REGION Network 21: bit gotowości wspólny Z9
   // AUMA
   // MODACT MOK250
   RUNG wire#powerrail
      Contact( "AlwaysTRUE" )
      Contact( "isPowerOK" )
      wire#w1
      Contact( "isAUMA_Z_9" )
      I_Contact( "inputAumagotowośćZ_9" )
      wire#w2
      R_Coil( "isGotowość_Z_9" )
   END_RUNG
   RUNG wire#w1
      Contact( "Hbit_Alarm_Z9" )
   END_RUNG wire#w2
   RUNG wire#w1
      I_Contact( "isAUMA_Z_9" )
      Contact( "setAlarm_Moment_Z_9" )
   END_RUNG wire#w2
   RUNG wire#w1
      Contact( "Hbit_Alarm_Z9" )
      Coil( "CMD_Awaria_Z_9" )
   END_RUNG
   // the same network as SCL:
   #_w1 := "AlwaysTRUE" AND "isPowerOK";
   IF #_w1 AND (("isAUMA_Z_9" AND NOT "inputAumagotowośćZ_9") OR "Hbit_Alarm_Z9" OR (NOT "isAUMA_Z_9" AND "setAlarm_Moment_Z_9")) THEN
       "isGotowość_Z_9" := FALSE;
   END_IF;
   "CMD_Awaria_Z_9" := #_w1 AND "Hbit_Alarm_Z9";
END_REGION
END_FUNCTION

FUNCTION "Wybór_aktywnego_zbiornika" : Void   // FC20, LAD
TITLE = Compressor selection from hours
{ S7_Optimized_Access := 'TRUE' }
AUTHOR : rtecmer
VERSION : 0.1
// Ustawienie kolejności wyboru zbiornika z wyrównaniem czasu pracy. Podstawa najmniejsza ilość godzin pracy
// stored: AutoNumber true, IsIECCheckEnabled false, SetENOAutomatically false, UDAEnableTagReadback false
   VAR_INPUT
      aktywny_Zbiornik_1 : Bool;   // zbiornik aktywny zasuwy na pozycji atomat
      aktywny_Zbiornik_2 : Bool;
      aktywny_Zbiornik_3 : Bool;
      aktywny_Zbiornik_4 : Bool;
      ready_Z1 : Bool;   // gotowość
      ready_Z2 : Bool;   // gotowość
      ready_Z3 : Bool;   // gotowość
      ready_Z4 : Bool;   // gotowość
      ready_Z5 : Bool;   // gotowość
      ready_Z6 : Bool;   // gotowość
      ready_Z7 : Bool;   // gotowość
      ready_Z8 : Bool;   // gotowość
      Is_Eptying : Bool;   // aktwny cykl napełniania
      Is_Filling : Bool;   // aktywny cykl pompownia
   END_VAR
   VAR_IN_OUT
      Reset : Bool;   // Reset po błędzie
      set_HWork_Tank_1 : Bool;   // ustawiony aktywny
      set_HWork_Tank_2 : Bool;   // ustawiony aktywny
      set_HWork_Tank_3 : Bool;   // ustawiony aktywny
      set_HWork_Tank_4 : Bool;   // ustawiony aktywny
      blok_tank_1 : Bool;   // blokowanie zbirnika w sekwencji
      blok_tank_2 : Bool;   // blokowanie zbirnika w sekwencji
      blok_tank_3 : Bool;   // blokowanie zbirnika w sekwencji
      blok_tank_4 : Bool;   // blokowanie zbirnika w sekwencji
   END_VAR
   VAR_TEMP
      tmp_Sum_sek_P1 : Real;
      tmp_Sum_sek_P2 : Real;
      tmp_Sum_sek_P3 : Real;
      tmp_Sum_sek_P4 : Real;
   END_VAR
BEGIN

REGION Network 1: Reakcja na równe liczniki
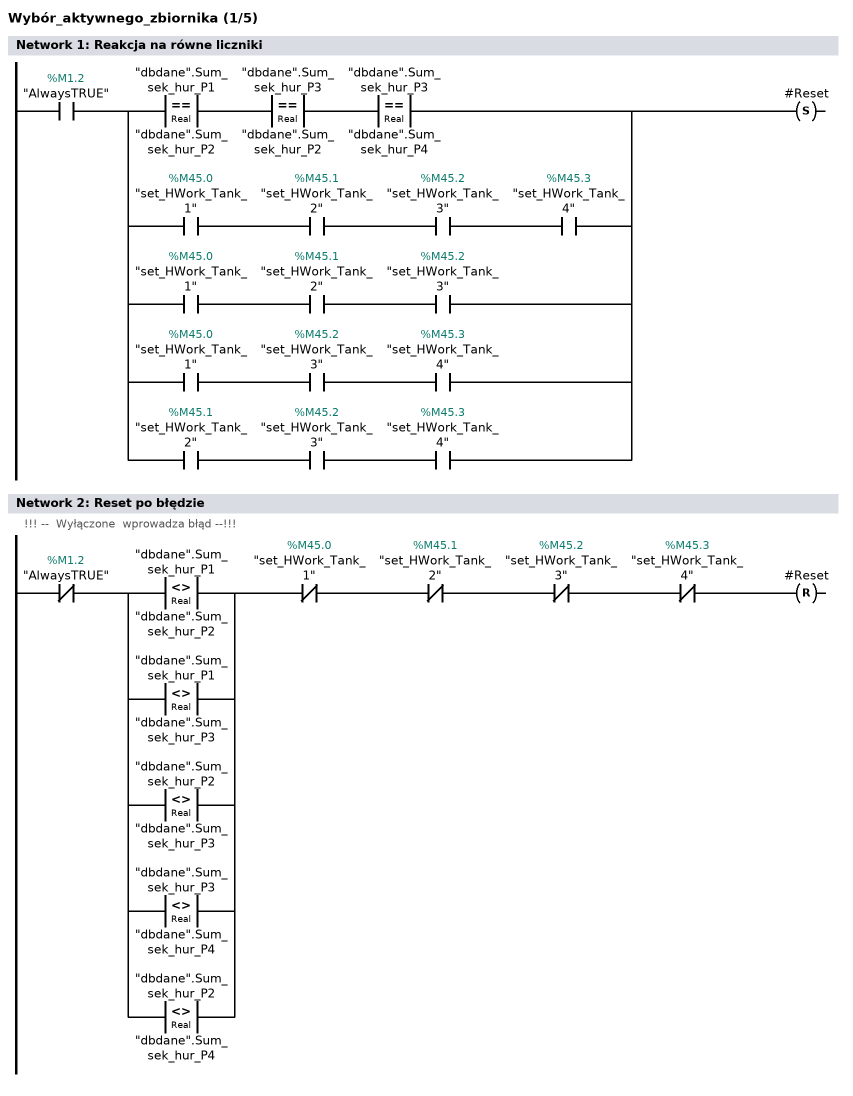
   RUNG wire#powerrail
      Contact( "AlwaysTRUE" )
      wire#w1
      { S7_Templates := "SrcType := Real" } EQ_Contact(in1 := "dbdane".Sum_sek_hur_P1, in2 := "dbdane".Sum_sek_hur_P2)
      { S7_Templates := "SrcType := Real" } EQ_Contact(in1 := "dbdane".Sum_sek_hur_P3, in2 := "dbdane".Sum_sek_hur_P2)
      { S7_Templates := "SrcType := Real" } EQ_Contact(in1 := "dbdane".Sum_sek_hur_P3, in2 := "dbdane".Sum_sek_hur_P4)
      wire#w2
      S_Coil( #Reset )
   END_RUNG
   RUNG wire#w1
      Contact( "set_HWork_Tank_1" )
      Contact( "set_HWork_Tank_2" )
      Contact( "set_HWork_Tank_3" )
      Contact( "set_HWork_Tank_4" )
   END_RUNG wire#w2
   RUNG wire#w1
      Contact( "set_HWork_Tank_1" )
      Contact( "set_HWork_Tank_2" )
      Contact( "set_HWork_Tank_3" )
   END_RUNG wire#w2
   RUNG wire#w1
      Contact( "set_HWork_Tank_1" )
      Contact( "set_HWork_Tank_3" )
      Contact( "set_HWork_Tank_4" )
   END_RUNG wire#w2
   RUNG wire#w1
      Contact( "set_HWork_Tank_2" )
      Contact( "set_HWork_Tank_3" )
      Contact( "set_HWork_Tank_4" )
   END_RUNG wire#w2
   // the same network as SCL:
   IF "AlwaysTRUE" AND ((("dbdane".Sum_sek_hur_P1 = "dbdane".Sum_sek_hur_P2) AND ("dbdane".Sum_sek_hur_P3 = "dbdane".Sum_sek_hur_P2) AND ("dbdane".Sum_sek_hur_P3 = "dbdane".Sum_sek_hur_P4)) OR ("set_HWork_Tank_1" AND "set_HWork_Tank_2" AND "set_HWork_Tank_3" AND "set_HWork_Tank_4") OR ("set_HWork_Tank_1" AND "set_HWork_Tank_2" AND "set_HWork_Tank_3") OR ("set_HWork_Tank_1" AND "set_HWork_Tank_3" AND "set_HWork_Tank_4") OR ("set_HWork_Tank_2" AND "set_HWork_Tank_3" AND "set_HWork_Tank_4")) THEN
       #Reset := TRUE;
   END_IF;
END_REGION

REGION Network 2: Reset po błędzie
   // !!! --  Wyłączone  wprowadza błąd --!!!
   RUNG wire#powerrail
      I_Contact( "AlwaysTRUE" )
      wire#w1
      { S7_Templates := "SrcType := Real" } NE_Contact(in1 := "dbdane".Sum_sek_hur_P1, in2 := "dbdane".Sum_sek_hur_P2)
      wire#w2
      I_Contact( "set_HWork_Tank_1" )
      I_Contact( "set_HWork_Tank_2" )
      I_Contact( "set_HWork_Tank_3" )
      I_Contact( "set_HWork_Tank_4" )
      R_Coil( #Reset )
   END_RUNG
   RUNG wire#w1
      { S7_Templates := "SrcType := Real" } NE_Contact(in1 := "dbdane".Sum_sek_hur_P1, in2 := "dbdane".Sum_sek_hur_P3)
   END_RUNG wire#w2
   RUNG wire#w1
      { S7_Templates := "SrcType := Real" } NE_Contact(in1 := "dbdane".Sum_sek_hur_P2, in2 := "dbdane".Sum_sek_hur_P3)
   END_RUNG wire#w2
   RUNG wire#w1
      { S7_Templates := "SrcType := Real" } NE_Contact(in1 := "dbdane".Sum_sek_hur_P3, in2 := "dbdane".Sum_sek_hur_P4)
   END_RUNG wire#w2
   RUNG wire#w1
      { S7_Templates := "SrcType := Real" } NE_Contact(in1 := "dbdane".Sum_sek_hur_P2, in2 := "dbdane".Sum_sek_hur_P4)
   END_RUNG wire#w2
   // the same network as SCL:
   IF NOT "AlwaysTRUE" AND (("dbdane".Sum_sek_hur_P1 <> "dbdane".Sum_sek_hur_P2) OR ("dbdane".Sum_sek_hur_P1 <> "dbdane".Sum_sek_hur_P3) OR ("dbdane".Sum_sek_hur_P2 <> "dbdane".Sum_sek_hur_P3) OR ("dbdane".Sum_sek_hur_P3 <> "dbdane".Sum_sek_hur_P4) OR ("dbdane".Sum_sek_hur_P2 <> "dbdane".Sum_sek_hur_P4)) AND NOT "set_HWork_Tank_1" AND NOT "set_HWork_Tank_2" AND NOT "set_HWork_Tank_3" AND NOT "set_HWork_Tank_4" THEN
       #Reset := FALSE;
   END_IF;
END_REGION

REGION Network 3: Wyłączenie napedów od równych liczników
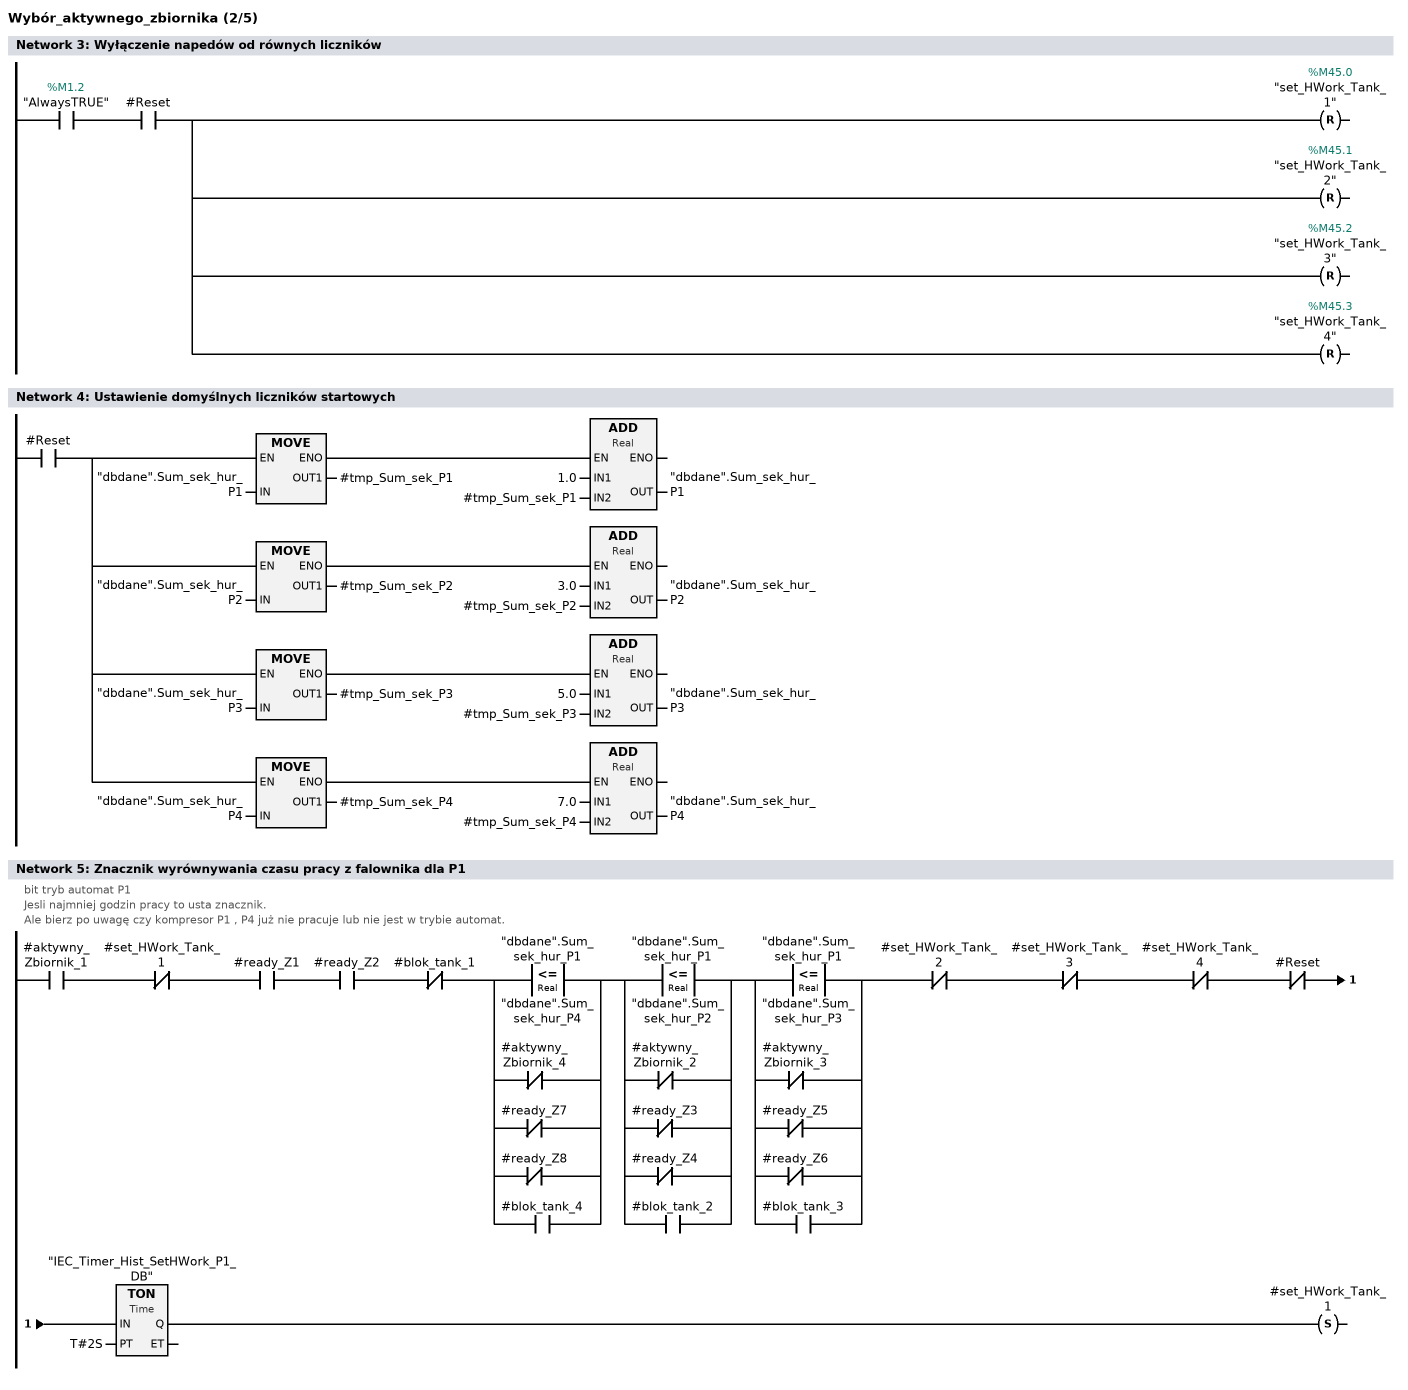
   RUNG wire#powerrail
      Contact( "AlwaysTRUE" )
      Contact( #Reset )
      wire#w1
      R_Coil( "set_HWork_Tank_1" )
   END_RUNG
   RUNG wire#w1
      R_Coil( "set_HWork_Tank_2" )
   END_RUNG
   RUNG wire#w1
      R_Coil( "set_HWork_Tank_3" )
   END_RUNG
   RUNG wire#w1
      R_Coil( "set_HWork_Tank_4" )
   END_RUNG
   // the same network as SCL:
   IF "AlwaysTRUE" AND #Reset THEN
       "set_HWork_Tank_1" := FALSE;
       "set_HWork_Tank_2" := FALSE;
       "set_HWork_Tank_3" := FALSE;
       "set_HWork_Tank_4" := FALSE;
   END_IF;
END_REGION

REGION Network 4: Ustawienie domyślnych liczników startowych
   RUNG wire#powerrail
      Contact( #Reset )
      wire#w1
      Move(in := "dbdane".Sum_sek_hur_P1, out1 => #tmp_Sum_sek_P1)
      { S7_Templates := "SrcType := Real" } Add(in1 := 1.0, in2 := #tmp_Sum_sek_P1, out => "dbdane".Sum_sek_hur_P1)
   END_RUNG
   RUNG wire#w1
      Move(in := "dbdane".Sum_sek_hur_P2, out1 => #tmp_Sum_sek_P2)
      { S7_Templates := "SrcType := Real" } Add(in1 := 3.0, in2 := #tmp_Sum_sek_P2, out => "dbdane".Sum_sek_hur_P2)
   END_RUNG
   RUNG wire#w1
      Move(in := "dbdane".Sum_sek_hur_P3, out1 => #tmp_Sum_sek_P3)
      { S7_Templates := "SrcType := Real" } Add(in1 := 5.0, in2 := #tmp_Sum_sek_P3, out => "dbdane".Sum_sek_hur_P3)
   END_RUNG
   RUNG wire#w1
      Move(in := "dbdane".Sum_sek_hur_P4, out1 => #tmp_Sum_sek_P4)
      { S7_Templates := "SrcType := Real" } Add(in1 := 7.0, in2 := #tmp_Sum_sek_P4, out => "dbdane".Sum_sek_hur_P4)
   END_RUNG
   // the same network as SCL:
   IF #Reset THEN
       #tmp_Sum_sek_P1 := "dbdane".Sum_sek_hur_P1;
       "dbdane".Sum_sek_hur_P1 := 1.0 + #tmp_Sum_sek_P1;
       #tmp_Sum_sek_P2 := "dbdane".Sum_sek_hur_P2;
       "dbdane".Sum_sek_hur_P2 := 3.0 + #tmp_Sum_sek_P2;
       #tmp_Sum_sek_P3 := "dbdane".Sum_sek_hur_P3;
       "dbdane".Sum_sek_hur_P3 := 5.0 + #tmp_Sum_sek_P3;
       #tmp_Sum_sek_P4 := "dbdane".Sum_sek_hur_P4;
       "dbdane".Sum_sek_hur_P4 := 7.0 + #tmp_Sum_sek_P4;
   END_IF;
END_REGION

REGION Network 5: Znacznik wyrównywania czasu pracy z falownika dla P1
   // bit tryb automat P1
   // Jesli najmniej godzin pracy to usta znacznik.
   // Ale bierz po uwagę czy kompresor P1 , P4 już nie pracuje lub nie jest w trybie automat.
   RUNG wire#powerrail
      Contact( #aktywny_Zbiornik_1 )
      I_Contact( #set_HWork_Tank_1 )
      Contact( #ready_Z1 )
      Contact( #ready_Z2 )
      I_Contact( #blok_tank_1 )
      wire#w1
      { S7_Templates := "SrcType := Real" } LE_Contact(in1 := "dbdane".Sum_sek_hur_P1, in2 := "dbdane".Sum_sek_hur_P4)
      wire#w2
      { S7_Templates := "SrcType := Real" } LE_Contact(in1 := "dbdane".Sum_sek_hur_P1, in2 := "dbdane".Sum_sek_hur_P2)
      wire#w3
      { S7_Templates := "SrcType := Real" } LE_Contact(in1 := "dbdane".Sum_sek_hur_P1, in2 := "dbdane".Sum_sek_hur_P3)
      wire#w4
      I_Contact( #set_HWork_Tank_2 )
      I_Contact( #set_HWork_Tank_3 )
      I_Contact( #set_HWork_Tank_4 )
      I_Contact( #Reset )
      { S7_Templates := "time_type := Time" } "IEC_Timer_Hist_SetHWork_P1_DB".TON(pt := T#2S, et =>)
      S_Coil( #set_HWork_Tank_1 )
   END_RUNG
   RUNG wire#w1
      I_Contact( #aktywny_Zbiornik_4 )
   END_RUNG wire#w2
   RUNG wire#w1
      I_Contact( #ready_Z7 )
   END_RUNG wire#w2
   RUNG wire#w1
      I_Contact( #ready_Z8 )
   END_RUNG wire#w2
   RUNG wire#w1
      Contact( #blok_tank_4 )
   END_RUNG wire#w2
   RUNG wire#w2
      I_Contact( #aktywny_Zbiornik_2 )
   END_RUNG wire#w3
   RUNG wire#w2
      I_Contact( #ready_Z3 )
   END_RUNG wire#w3
   RUNG wire#w2
      I_Contact( #ready_Z4 )
   END_RUNG wire#w3
   RUNG wire#w2
      Contact( #blok_tank_2 )
   END_RUNG wire#w3
   RUNG wire#w3
      I_Contact( #aktywny_Zbiornik_3 )
   END_RUNG wire#w4
   RUNG wire#w3
      I_Contact( #ready_Z5 )
   END_RUNG wire#w4
   RUNG wire#w3
      I_Contact( #ready_Z6 )
   END_RUNG wire#w4
   RUNG wire#w3
      Contact( #blok_tank_3 )
   END_RUNG wire#w4
   // the same network as SCL:
   "IEC_Timer_Hist_SetHWork_P1_DB".TON(IN := #aktywny_Zbiornik_1 AND NOT #set_HWork_Tank_1 AND #ready_Z1 AND #ready_Z2 AND NOT #blok_tank_1 AND (("dbdane".Sum_sek_hur_P1 <= "dbdane".Sum_sek_hur_P4) OR NOT #aktywny_Zbiornik_4 OR NOT #ready_Z7 OR NOT #ready_Z8 OR #blok_tank_4) AND (("dbdane".Sum_sek_hur_P1 <= "dbdane".Sum_sek_hur_P2) OR NOT #aktywny_Zbiornik_2 OR NOT #ready_Z3 OR NOT #ready_Z4 OR #blok_tank_2) AND (("dbdane".Sum_sek_hur_P1 <= "dbdane".Sum_sek_hur_P3) OR NOT #aktywny_Zbiornik_3 OR NOT #ready_Z5 OR NOT #ready_Z6 OR #blok_tank_3) AND NOT #set_HWork_Tank_2 AND NOT #set_HWork_Tank_3 AND NOT #set_HWork_Tank_4 AND NOT #Reset,
                           PT := T#2S);
   IF "IEC_Timer_Hist_SetHWork_P1_DB".Q THEN #set_HWork_Tank_1 := TRUE; END_IF;
END_REGION

REGION Network 6 (SCL): Sprawdzanie czy aktywna w trybie AUT
   IF "set_HWork_Tank_1" = TRUE AND #aktywny_Zbiornik_1 = FALSE THEN
     // Statement section IF
     "set_HWork_Tank_1" := FALSE;
     ;
   END_IF;
END_REGION

REGION Network 7: Znacznik ustawienia pracy od licznika pracy P1
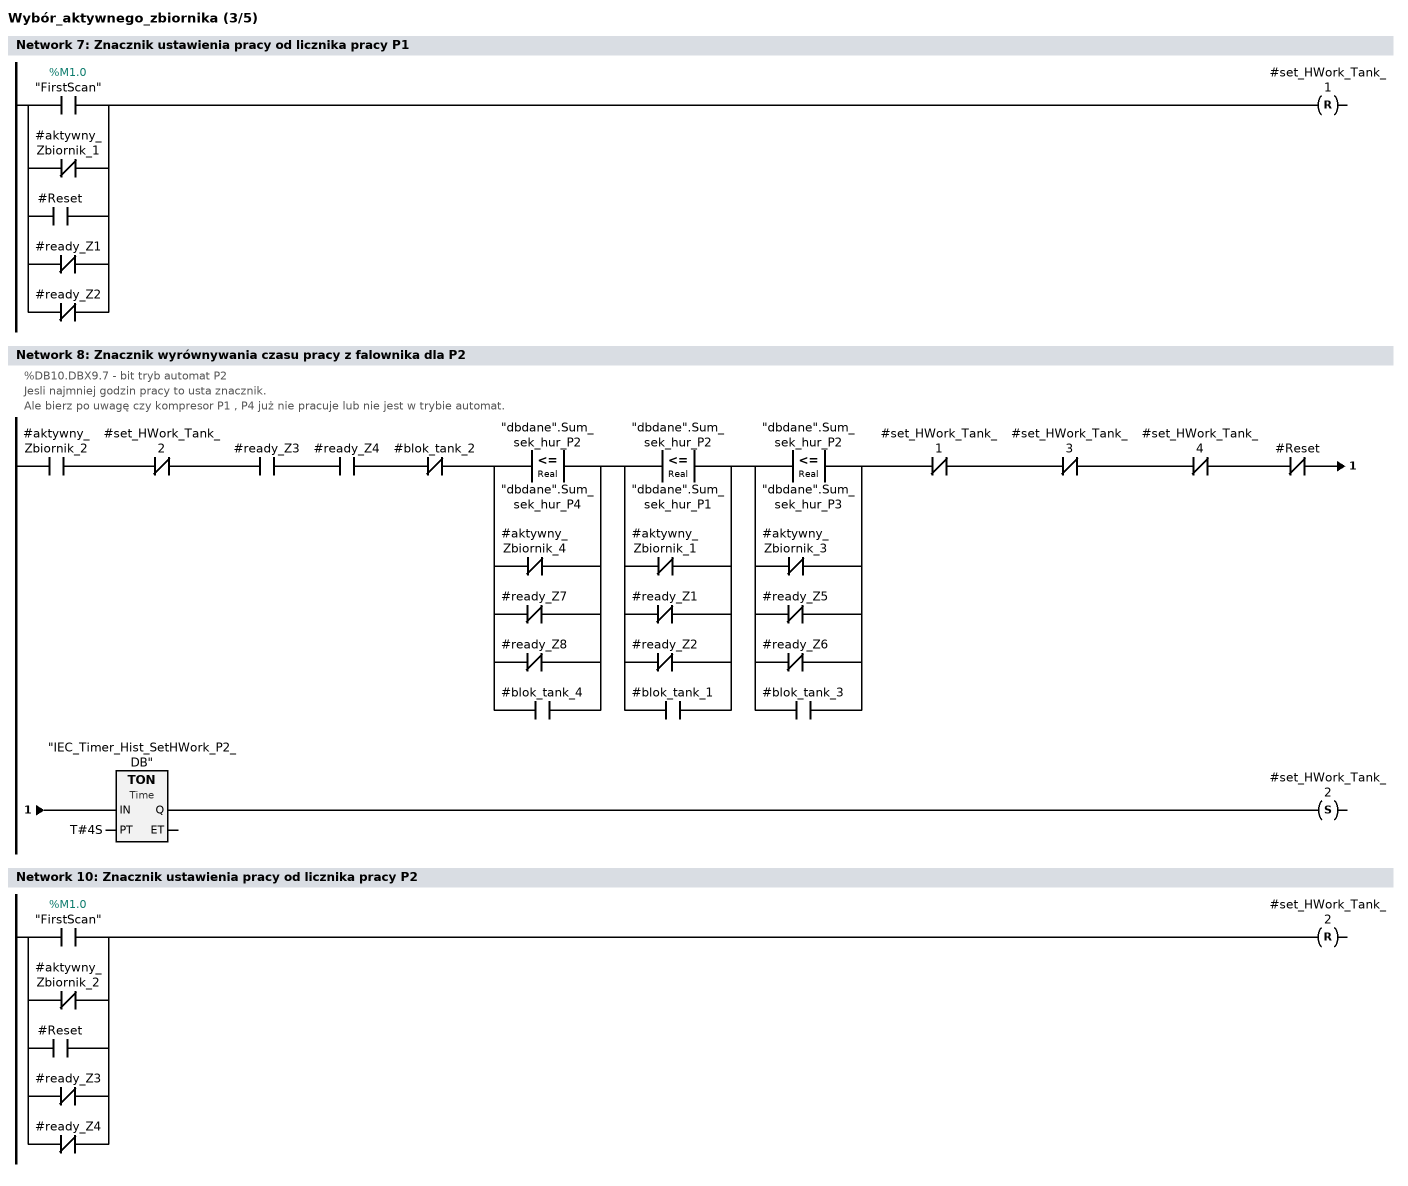
   RUNG wire#powerrail
      Contact( "FirstScan" )
      wire#w1
      R_Coil( #set_HWork_Tank_1 )
   END_RUNG
   RUNG wire#powerrail
      I_Contact( #aktywny_Zbiornik_1 )
   END_RUNG wire#w1
   RUNG wire#powerrail
      Contact( #Reset )
   END_RUNG wire#w1
   RUNG wire#powerrail
      I_Contact( #ready_Z1 )
   END_RUNG wire#w1
   RUNG wire#powerrail
      I_Contact( #ready_Z2 )
   END_RUNG wire#w1
   // the same network as SCL:
   IF "FirstScan" OR NOT #aktywny_Zbiornik_1 OR #Reset OR NOT #ready_Z1 OR NOT #ready_Z2 THEN
       #set_HWork_Tank_1 := FALSE;
   END_IF;
END_REGION

REGION Network 8: Znacznik wyrównywania czasu pracy z falownika dla P2
   // %DB10.DBX9.7 - bit tryb automat P2
   // Jesli najmniej godzin pracy to usta znacznik.
   // Ale bierz po uwagę czy kompresor P1 , P4 już nie pracuje lub nie jest w trybie automat.
   RUNG wire#powerrail
      Contact( #aktywny_Zbiornik_2 )
      I_Contact( #set_HWork_Tank_2 )
      Contact( #ready_Z3 )
      Contact( #ready_Z4 )
      I_Contact( #blok_tank_2 )
      wire#w1
      { S7_Templates := "SrcType := Real" } LE_Contact(in1 := "dbdane".Sum_sek_hur_P2, in2 := "dbdane".Sum_sek_hur_P4)
      wire#w2
      { S7_Templates := "SrcType := Real" } LE_Contact(in1 := "dbdane".Sum_sek_hur_P2, in2 := "dbdane".Sum_sek_hur_P1)
      wire#w3
      { S7_Templates := "SrcType := Real" } LE_Contact(in1 := "dbdane".Sum_sek_hur_P2, in2 := "dbdane".Sum_sek_hur_P3)
      wire#w4
      I_Contact( #set_HWork_Tank_1 )
      I_Contact( #set_HWork_Tank_3 )
      I_Contact( #set_HWork_Tank_4 )
      I_Contact( #Reset )
      { S7_Templates := "time_type := Time" } "IEC_Timer_Hist_SetHWork_P2_DB".TON(pt := T#4S, et =>)
      S_Coil( #set_HWork_Tank_2 )
   END_RUNG
   RUNG wire#w1
      I_Contact( #aktywny_Zbiornik_4 )
   END_RUNG wire#w2
   RUNG wire#w1
      I_Contact( #ready_Z7 )
   END_RUNG wire#w2
   RUNG wire#w1
      I_Contact( #ready_Z8 )
   END_RUNG wire#w2
   RUNG wire#w1
      Contact( #blok_tank_4 )
   END_RUNG wire#w2
   RUNG wire#w2
      I_Contact( #aktywny_Zbiornik_1 )
   END_RUNG wire#w3
   RUNG wire#w2
      I_Contact( #ready_Z1 )
   END_RUNG wire#w3
   RUNG wire#w2
      I_Contact( #ready_Z2 )
   END_RUNG wire#w3
   RUNG wire#w2
      Contact( #blok_tank_1 )
   END_RUNG wire#w3
   RUNG wire#w3
      I_Contact( #aktywny_Zbiornik_3 )
   END_RUNG wire#w4
   RUNG wire#w3
      I_Contact( #ready_Z5 )
   END_RUNG wire#w4
   RUNG wire#w3
      I_Contact( #ready_Z6 )
   END_RUNG wire#w4
   RUNG wire#w3
      Contact( #blok_tank_3 )
   END_RUNG wire#w4
   // the same network as SCL:
   "IEC_Timer_Hist_SetHWork_P2_DB".TON(IN := #aktywny_Zbiornik_2 AND NOT #set_HWork_Tank_2 AND #ready_Z3 AND #ready_Z4 AND NOT #blok_tank_2 AND (("dbdane".Sum_sek_hur_P2 <= "dbdane".Sum_sek_hur_P4) OR NOT #aktywny_Zbiornik_4 OR NOT #ready_Z7 OR NOT #ready_Z8 OR #blok_tank_4) AND (("dbdane".Sum_sek_hur_P2 <= "dbdane".Sum_sek_hur_P1) OR NOT #aktywny_Zbiornik_1 OR NOT #ready_Z1 OR NOT #ready_Z2 OR #blok_tank_1) AND (("dbdane".Sum_sek_hur_P2 <= "dbdane".Sum_sek_hur_P3) OR NOT #aktywny_Zbiornik_3 OR NOT #ready_Z5 OR NOT #ready_Z6 OR #blok_tank_3) AND NOT #set_HWork_Tank_1 AND NOT #set_HWork_Tank_3 AND NOT #set_HWork_Tank_4 AND NOT #Reset,
                           PT := T#4S);
   IF "IEC_Timer_Hist_SetHWork_P2_DB".Q THEN #set_HWork_Tank_2 := TRUE; END_IF;
END_REGION

REGION Network 9 (SCL): Sprawdzanie czy aktywna w trybie AUT
   IF "set_HWork_Tank_2" = TRUE AND #aktywny_Zbiornik_2 = FALSE THEN
     // Statement section IF
     "set_HWork_Tank_2" := FALSE;
     ;
   END_IF;
END_REGION

REGION Network 10: Znacznik ustawienia pracy od licznika pracy P2
   RUNG wire#powerrail
      Contact( "FirstScan" )
      wire#w1
      R_Coil( #set_HWork_Tank_2 )
   END_RUNG
   RUNG wire#powerrail
      I_Contact( #aktywny_Zbiornik_2 )
   END_RUNG wire#w1
   RUNG wire#powerrail
      Contact( #Reset )
   END_RUNG wire#w1
   RUNG wire#powerrail
      I_Contact( #ready_Z3 )
   END_RUNG wire#w1
   RUNG wire#powerrail
      I_Contact( #ready_Z4 )
   END_RUNG wire#w1
   // the same network as SCL:
   IF "FirstScan" OR NOT #aktywny_Zbiornik_2 OR #Reset OR NOT #ready_Z3 OR NOT #ready_Z4 THEN
       #set_HWork_Tank_2 := FALSE;
   END_IF;
END_REGION

REGION Network 11: Znacznik wyrównywania czasu pracy z falownika P3
   // bit tryb automat P3
   // Jesli najmniej godzin pracy to usta znacznik.
   // Ale bierz po uwagę czy P1, P4 już nie pracuje lub nie jest w trybie automat.
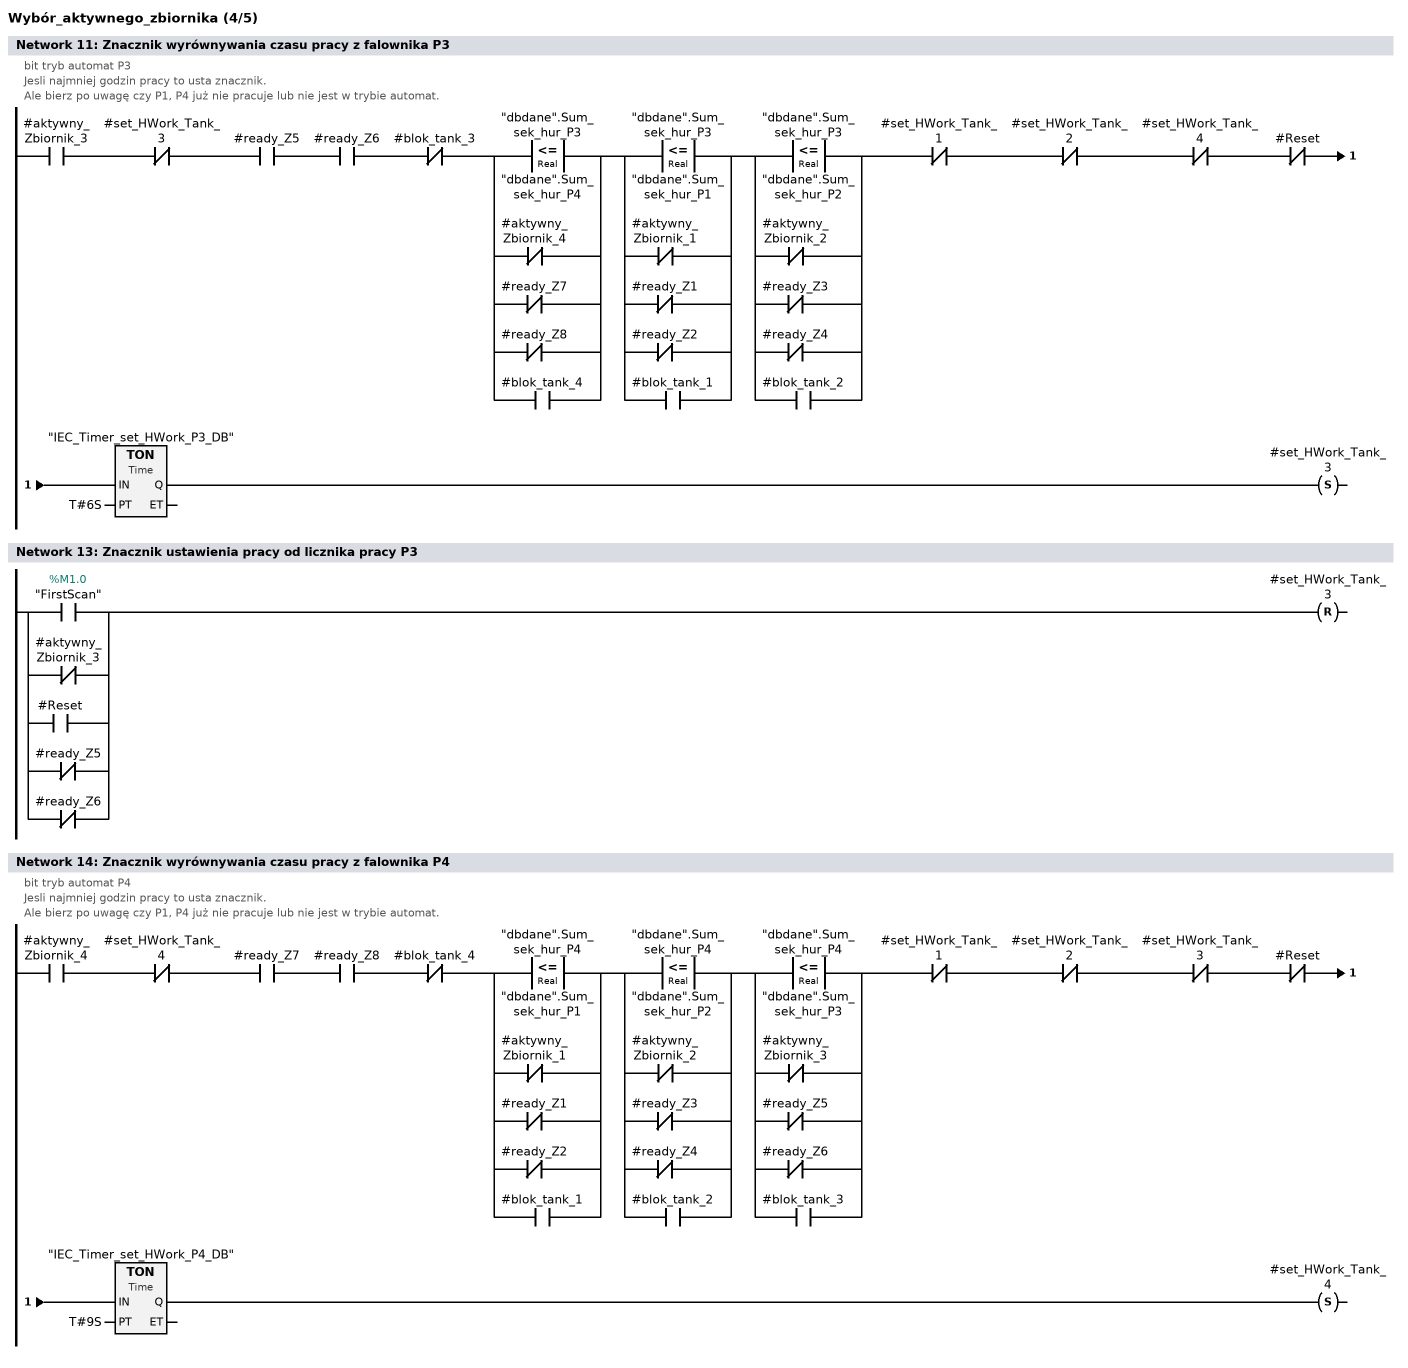
   RUNG wire#powerrail
      Contact( #aktywny_Zbiornik_3 )
      I_Contact( #set_HWork_Tank_3 )
      Contact( #ready_Z5 )
      Contact( #ready_Z6 )
      I_Contact( #blok_tank_3 )
      wire#w1
      { S7_Templates := "SrcType := Real" } LE_Contact(in1 := "dbdane".Sum_sek_hur_P3, in2 := "dbdane".Sum_sek_hur_P4)
      wire#w2
      { S7_Templates := "SrcType := Real" } LE_Contact(in1 := "dbdane".Sum_sek_hur_P3, in2 := "dbdane".Sum_sek_hur_P1)
      wire#w3
      { S7_Templates := "SrcType := Real" } LE_Contact(in1 := "dbdane".Sum_sek_hur_P3, in2 := "dbdane".Sum_sek_hur_P2)
      wire#w4
      I_Contact( #set_HWork_Tank_1 )
      I_Contact( #set_HWork_Tank_2 )
      I_Contact( #set_HWork_Tank_4 )
      I_Contact( #Reset )
      { S7_Templates := "time_type := Time" } "IEC_Timer_set_HWork_P3_DB".TON(pt := T#6S, et =>)
      S_Coil( #set_HWork_Tank_3 )
   END_RUNG
   RUNG wire#w1
      I_Contact( #aktywny_Zbiornik_4 )
   END_RUNG wire#w2
   RUNG wire#w1
      I_Contact( #ready_Z7 )
   END_RUNG wire#w2
   RUNG wire#w1
      I_Contact( #ready_Z8 )
   END_RUNG wire#w2
   RUNG wire#w1
      Contact( #blok_tank_4 )
   END_RUNG wire#w2
   RUNG wire#w2
      I_Contact( #aktywny_Zbiornik_1 )
   END_RUNG wire#w3
   RUNG wire#w2
      I_Contact( #ready_Z1 )
   END_RUNG wire#w3
   RUNG wire#w2
      I_Contact( #ready_Z2 )
   END_RUNG wire#w3
   RUNG wire#w2
      Contact( #blok_tank_1 )
   END_RUNG wire#w3
   RUNG wire#w3
      I_Contact( #aktywny_Zbiornik_2 )
   END_RUNG wire#w4
   RUNG wire#w3
      I_Contact( #ready_Z3 )
   END_RUNG wire#w4
   RUNG wire#w3
      I_Contact( #ready_Z4 )
   END_RUNG wire#w4
   RUNG wire#w3
      Contact( #blok_tank_2 )
   END_RUNG wire#w4
   // the same network as SCL:
   "IEC_Timer_set_HWork_P3_DB".TON(IN := #aktywny_Zbiornik_3 AND NOT #set_HWork_Tank_3 AND #ready_Z5 AND #ready_Z6 AND NOT #blok_tank_3 AND (("dbdane".Sum_sek_hur_P3 <= "dbdane".Sum_sek_hur_P4) OR NOT #aktywny_Zbiornik_4 OR NOT #ready_Z7 OR NOT #ready_Z8 OR #blok_tank_4) AND (("dbdane".Sum_sek_hur_P3 <= "dbdane".Sum_sek_hur_P1) OR NOT #aktywny_Zbiornik_1 OR NOT #ready_Z1 OR NOT #ready_Z2 OR #blok_tank_1) AND (("dbdane".Sum_sek_hur_P3 <= "dbdane".Sum_sek_hur_P2) OR NOT #aktywny_Zbiornik_2 OR NOT #ready_Z3 OR NOT #ready_Z4 OR #blok_tank_2) AND NOT #set_HWork_Tank_1 AND NOT #set_HWork_Tank_2 AND NOT #set_HWork_Tank_4 AND NOT #Reset,
                           PT := T#6S);
   IF "IEC_Timer_set_HWork_P3_DB".Q THEN #set_HWork_Tank_3 := TRUE; END_IF;
END_REGION

REGION Network 12 (SCL): Sprawdzanie czy aktywna w trybie AUT
   IF "set_HWork_Tank_3" = TRUE AND #aktywny_Zbiornik_3 = FALSE THEN
     // Statement section IF
     "set_HWork_Tank_3":= FALSE;
     ;
   END_IF;
END_REGION

REGION Network 13: Znacznik ustawienia pracy od licznika pracy P3
   RUNG wire#powerrail
      Contact( "FirstScan" )
      wire#w1
      R_Coil( #set_HWork_Tank_3 )
   END_RUNG
   RUNG wire#powerrail
      I_Contact( #aktywny_Zbiornik_3 )
   END_RUNG wire#w1
   RUNG wire#powerrail
      Contact( #Reset )
   END_RUNG wire#w1
   RUNG wire#powerrail
      I_Contact( #ready_Z5 )
   END_RUNG wire#w1
   RUNG wire#powerrail
      I_Contact( #ready_Z6 )
   END_RUNG wire#w1
   // the same network as SCL:
   IF "FirstScan" OR NOT #aktywny_Zbiornik_3 OR #Reset OR NOT #ready_Z5 OR NOT #ready_Z6 THEN
       #set_HWork_Tank_3 := FALSE;
   END_IF;
END_REGION

REGION Network 14: Znacznik wyrównywania czasu pracy z falownika P4
   // bit tryb automat P4
   // Jesli najmniej godzin pracy to usta znacznik.
   // Ale bierz po uwagę czy P1, P4 już nie pracuje lub nie jest w trybie automat.
   RUNG wire#powerrail
      Contact( #aktywny_Zbiornik_4 )
      I_Contact( #set_HWork_Tank_4 )
      Contact( #ready_Z7 )
      Contact( #ready_Z8 )
      I_Contact( #blok_tank_4 )
      wire#w1
      { S7_Templates := "SrcType := Real" } LE_Contact(in1 := "dbdane".Sum_sek_hur_P4, in2 := "dbdane".Sum_sek_hur_P1)
      wire#w2
      { S7_Templates := "SrcType := Real" } LE_Contact(in1 := "dbdane".Sum_sek_hur_P4, in2 := "dbdane".Sum_sek_hur_P2)
      wire#w3
      { S7_Templates := "SrcType := Real" } LE_Contact(in1 := "dbdane".Sum_sek_hur_P4, in2 := "dbdane".Sum_sek_hur_P3)
      wire#w4
      I_Contact( #set_HWork_Tank_1 )
      I_Contact( #set_HWork_Tank_2 )
      I_Contact( #set_HWork_Tank_3 )
      I_Contact( #Reset )
      { S7_Templates := "time_type := Time" } "IEC_Timer_set_HWork_P4_DB".TON(pt := T#9S, et =>)
      S_Coil( #set_HWork_Tank_4 )
   END_RUNG
   RUNG wire#w1
      I_Contact( #aktywny_Zbiornik_1 )
   END_RUNG wire#w2
   RUNG wire#w1
      I_Contact( #ready_Z1 )
   END_RUNG wire#w2
   RUNG wire#w1
      I_Contact( #ready_Z2 )
   END_RUNG wire#w2
   RUNG wire#w1
      Contact( #blok_tank_1 )
   END_RUNG wire#w2
   RUNG wire#w2
      I_Contact( #aktywny_Zbiornik_2 )
   END_RUNG wire#w3
   RUNG wire#w2
      I_Contact( #ready_Z3 )
   END_RUNG wire#w3
   RUNG wire#w2
      I_Contact( #ready_Z4 )
   END_RUNG wire#w3
   RUNG wire#w2
      Contact( #blok_tank_2 )
   END_RUNG wire#w3
   RUNG wire#w3
      I_Contact( #aktywny_Zbiornik_3 )
   END_RUNG wire#w4
   RUNG wire#w3
      I_Contact( #ready_Z5 )
   END_RUNG wire#w4
   RUNG wire#w3
      I_Contact( #ready_Z6 )
   END_RUNG wire#w4
   RUNG wire#w3
      Contact( #blok_tank_3 )
   END_RUNG wire#w4
   // the same network as SCL:
   "IEC_Timer_set_HWork_P4_DB".TON(IN := #aktywny_Zbiornik_4 AND NOT #set_HWork_Tank_4 AND #ready_Z7 AND #ready_Z8 AND NOT #blok_tank_4 AND (("dbdane".Sum_sek_hur_P4 <= "dbdane".Sum_sek_hur_P1) OR NOT #aktywny_Zbiornik_1 OR NOT #ready_Z1 OR NOT #ready_Z2 OR #blok_tank_1) AND (("dbdane".Sum_sek_hur_P4 <= "dbdane".Sum_sek_hur_P2) OR NOT #aktywny_Zbiornik_2 OR NOT #ready_Z3 OR NOT #ready_Z4 OR #blok_tank_2) AND (("dbdane".Sum_sek_hur_P4 <= "dbdane".Sum_sek_hur_P3) OR NOT #aktywny_Zbiornik_3 OR NOT #ready_Z5 OR NOT #ready_Z6 OR #blok_tank_3) AND NOT #set_HWork_Tank_1 AND NOT #set_HWork_Tank_2 AND NOT #set_HWork_Tank_3 AND NOT #Reset,
                           PT := T#9S);
   IF "IEC_Timer_set_HWork_P4_DB".Q THEN #set_HWork_Tank_4 := TRUE; END_IF;
END_REGION

REGION Network 15 (SCL): Sprawdzanie czy aktywna w trybie AUT
   IF "set_HWork_Tank_4" = TRUE AND #aktywny_Zbiornik_4 = FALSE THEN
     // Statement section IF
     "set_HWork_Tank_4" := FALSE;
     ;
   END_IF;
END_REGION

REGION Network 16: Znacznik ustawienia pracy od licznika pracy P4
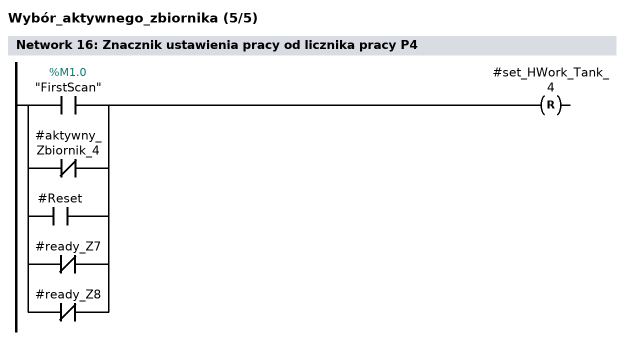
   RUNG wire#powerrail
      Contact( "FirstScan" )
      wire#w1
      R_Coil( #set_HWork_Tank_4 )
   END_RUNG
   RUNG wire#powerrail
      I_Contact( #aktywny_Zbiornik_4 )
   END_RUNG wire#w1
   RUNG wire#powerrail
      Contact( #Reset )
   END_RUNG wire#w1
   RUNG wire#powerrail
      I_Contact( #ready_Z7 )
   END_RUNG wire#w1
   RUNG wire#powerrail
      I_Contact( #ready_Z8 )
   END_RUNG wire#w1
   // the same network as SCL:
   IF "FirstScan" OR NOT #aktywny_Zbiornik_4 OR #Reset OR NOT #ready_Z7 OR NOT #ready_Z8 THEN
       #set_HWork_Tank_4 := FALSE;
   END_IF;
END_REGION
END_FUNCTION

FUNCTION_BLOCK "Startegia_sterowania"   // FB18, LAD
TITLE = Strategia przełączania
{ S7_Optimized_Access := 'TRUE' }
AUTHOR : rtecmer
VERSION : 0.1
// Funkcja przełącza stan aktywnego zbiornika w trybie napełniania i opróróżniana. Cykl pracy . Zbiornik opróżniany zostaje aktywny do napełniania a jeden pełny aktywny do przetłaczannia. 
// Znacznik blok_tank_x - blukuje zbiornik po zakonczonym cyklu do czasu aż wszystkie zbiorniki nie przejdą sekwencji.
// stored: AutoNumber true, IsIECCheckEnabled false, IsRetainMemResEnabled false, MemoryReserve 250, SetENOAutomatically false, UDAEnableTagReadback false
   VAR
      tmp_time_1 : Bool;   // pomocniczy bit do wyzwolenia opóźnionego resetu aktywnego zbiornika
      tmp_time_2 : Bool := false;   // pomocniczy bit do wyzwolenia opóźnionego resetu aktywnego zbiornika
      tmp_time_3 : Bool := false;   // pomocniczy bit do wyzwolenia opóźnionego resetu aktywnego zbiornika
      tmp_time_4 : Bool := false;   // pomocniczy bit do wyzwolenia opóźnionego resetu aktywnego zbiornika
   END_VAR
   VAR_TEMP   // added for the SCL form of the ladder/FBD networks
      _w1 : Bool;
      _w2 : Bool;
   END_VAR
BEGIN

REGION Network 2: jest zablokowany po pracy w sekwencji
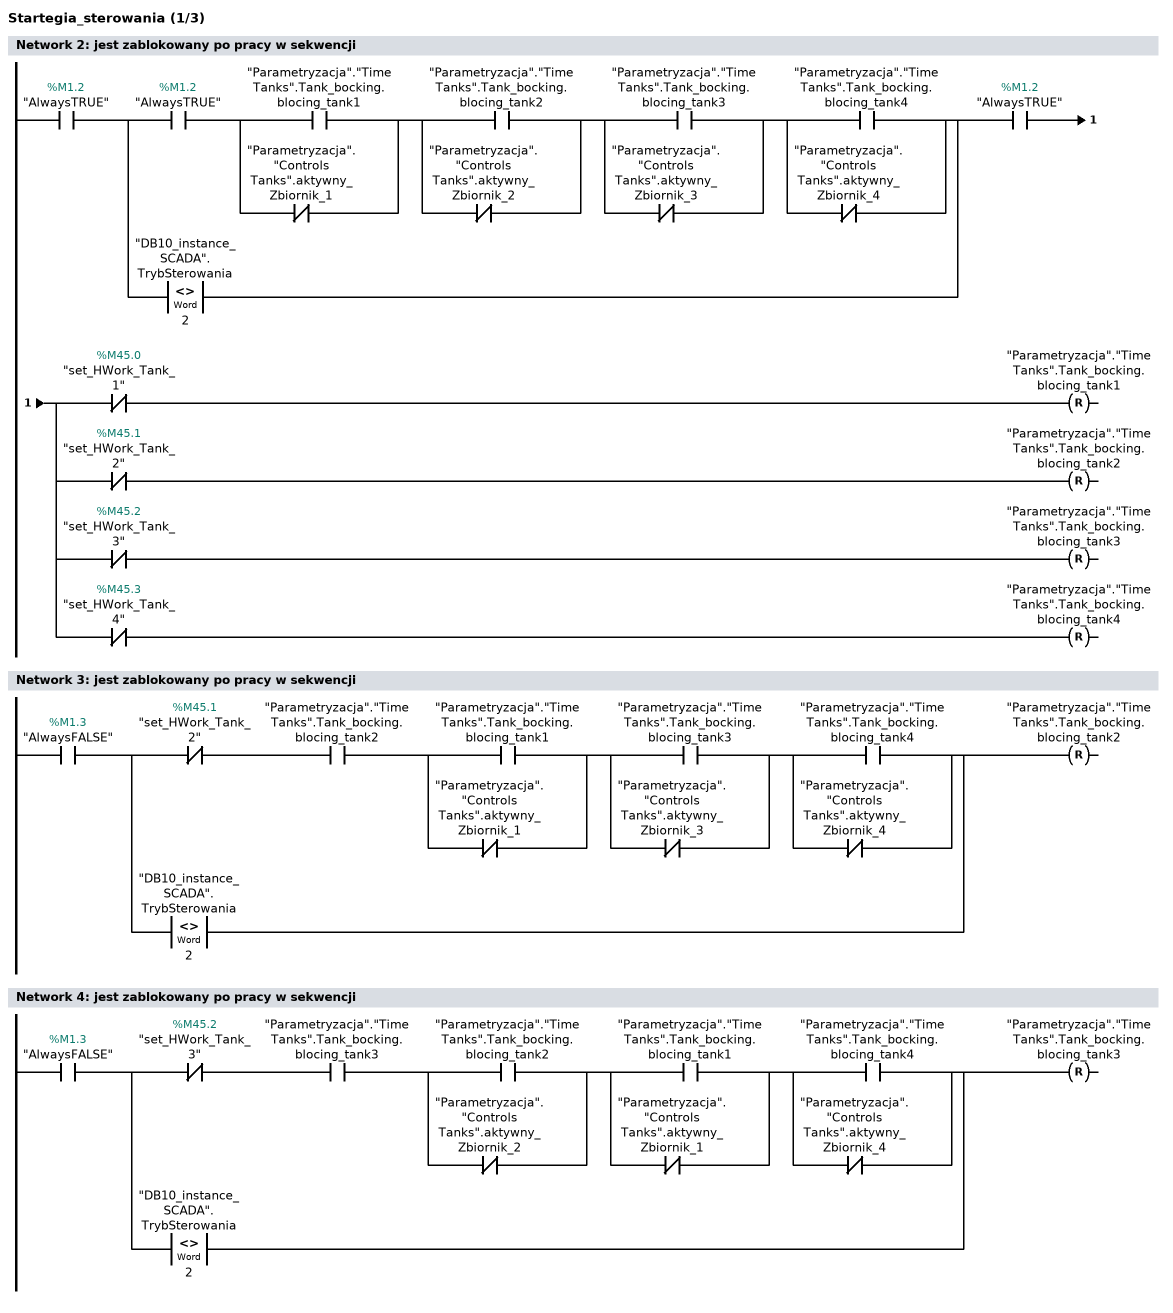
   RUNG wire#powerrail
      Contact( "AlwaysTRUE" )
      wire#w1
      Contact( "AlwaysTRUE" )
      wire#w2
      Contact( "Parametryzacja"."Time Tanks".Tank_bocking.blocing_tank1 )
      wire#w3
      Contact( "Parametryzacja"."Time Tanks".Tank_bocking.blocing_tank2 )
      wire#w4
      Contact( "Parametryzacja"."Time Tanks".Tank_bocking.blocing_tank3 )
      wire#w5
      Contact( "Parametryzacja"."Time Tanks".Tank_bocking.blocing_tank4 )
      wire#w6
      Contact( "AlwaysTRUE" )
      wire#w7
      I_Contact( "set_HWork_Tank_1" )
      R_Coil( "Parametryzacja"."Time Tanks".Tank_bocking.blocing_tank1 )
   END_RUNG
   RUNG wire#w2
      I_Contact( "Parametryzacja"."Controls Tanks".aktywny_Zbiornik_1 )
   END_RUNG wire#w3
   RUNG wire#w3
      I_Contact( "Parametryzacja"."Controls Tanks".aktywny_Zbiornik_2 )
   END_RUNG wire#w4
   RUNG wire#w4
      I_Contact( "Parametryzacja"."Controls Tanks".aktywny_Zbiornik_3 )
   END_RUNG wire#w5
   RUNG wire#w5
      I_Contact( "Parametryzacja"."Controls Tanks".aktywny_Zbiornik_4 )
   END_RUNG wire#w6
   RUNG wire#w1
      { S7_Templates := "SrcType := Word" } NE_Contact(in1 := "DB10_instance_SCADA".TrybSterowania, in2 := 2)
   END_RUNG wire#w6
   RUNG wire#w7
      I_Contact( "set_HWork_Tank_2" )
      R_Coil( "Parametryzacja"."Time Tanks".Tank_bocking.blocing_tank2 )
   END_RUNG
   RUNG wire#w7
      I_Contact( "set_HWork_Tank_3" )
      R_Coil( "Parametryzacja"."Time Tanks".Tank_bocking.blocing_tank3 )
   END_RUNG
   RUNG wire#w7
      I_Contact( "set_HWork_Tank_4" )
      R_Coil( "Parametryzacja"."Time Tanks".Tank_bocking.blocing_tank4 )
   END_RUNG
   // the same network as SCL:
   #_w1 := "AlwaysTRUE" AND (("AlwaysTRUE" AND ("Parametryzacja"."Time Tanks".Tank_bocking.blocing_tank1 OR NOT "Parametryzacja"."Controls Tanks".aktywny_Zbiornik_1) AND ("Parametryzacja"."Time Tanks".Tank_bocking.blocing_tank2 OR NOT "Parametryzacja"."Controls Tanks".aktywny_Zbiornik_2) AND ("Parametryzacja"."Time Tanks".Tank_bocking.blocing_tank3 OR NOT "Parametryzacja"."Controls Tanks".aktywny_Zbiornik_3) AND ("Parametryzacja"."Time Tanks".Tank_bocking.blocing_tank4 OR NOT "Parametryzacja"."Controls Tanks".aktywny_Zbiornik_4)) OR ("DB10_instance_SCADA".TrybSterowania <> 2)) AND "AlwaysTRUE";
   IF #_w1 AND NOT "set_HWork_Tank_1" THEN
       "Parametryzacja"."Time Tanks".Tank_bocking.blocing_tank1 := FALSE;
   END_IF;
   IF #_w1 AND NOT "set_HWork_Tank_2" THEN
       "Parametryzacja"."Time Tanks".Tank_bocking.blocing_tank2 := FALSE;
   END_IF;
   IF #_w1 AND NOT "set_HWork_Tank_3" THEN
       "Parametryzacja"."Time Tanks".Tank_bocking.blocing_tank3 := FALSE;
   END_IF;
   IF #_w1 AND NOT "set_HWork_Tank_4" THEN
       "Parametryzacja"."Time Tanks".Tank_bocking.blocing_tank4 := FALSE;
   END_IF;
END_REGION

REGION Network 3: jest zablokowany po pracy w sekwencji
   RUNG wire#powerrail
      Contact( "AlwaysFALSE" )
      wire#w1
      I_Contact( "set_HWork_Tank_2" )
      Contact( "Parametryzacja"."Time Tanks".Tank_bocking.blocing_tank2 )
      wire#w2
      Contact( "Parametryzacja"."Time Tanks".Tank_bocking.blocing_tank1 )
      wire#w3
      Contact( "Parametryzacja"."Time Tanks".Tank_bocking.blocing_tank3 )
      wire#w4
      Contact( "Parametryzacja"."Time Tanks".Tank_bocking.blocing_tank4 )
      wire#w5
      R_Coil( "Parametryzacja"."Time Tanks".Tank_bocking.blocing_tank2 )
   END_RUNG
   RUNG wire#w2
      I_Contact( "Parametryzacja"."Controls Tanks".aktywny_Zbiornik_1 )
   END_RUNG wire#w3
   RUNG wire#w3
      I_Contact( "Parametryzacja"."Controls Tanks".aktywny_Zbiornik_3 )
   END_RUNG wire#w4
   RUNG wire#w4
      I_Contact( "Parametryzacja"."Controls Tanks".aktywny_Zbiornik_4 )
   END_RUNG wire#w5
   RUNG wire#w1
      { S7_Templates := "SrcType := Word" } NE_Contact(in1 := "DB10_instance_SCADA".TrybSterowania, in2 := 2)
   END_RUNG wire#w5
   // the same network as SCL:
   IF "AlwaysFALSE" AND ((NOT "set_HWork_Tank_2" AND "Parametryzacja"."Time Tanks".Tank_bocking.blocing_tank2 AND ("Parametryzacja"."Time Tanks".Tank_bocking.blocing_tank1 OR NOT "Parametryzacja"."Controls Tanks".aktywny_Zbiornik_1) AND ("Parametryzacja"."Time Tanks".Tank_bocking.blocing_tank3 OR NOT "Parametryzacja"."Controls Tanks".aktywny_Zbiornik_3) AND ("Parametryzacja"."Time Tanks".Tank_bocking.blocing_tank4 OR NOT "Parametryzacja"."Controls Tanks".aktywny_Zbiornik_4)) OR ("DB10_instance_SCADA".TrybSterowania <> 2)) THEN
       "Parametryzacja"."Time Tanks".Tank_bocking.blocing_tank2 := FALSE;
   END_IF;
END_REGION

REGION Network 4: jest zablokowany po pracy w sekwencji
   RUNG wire#powerrail
      Contact( "AlwaysFALSE" )
      wire#w1
      I_Contact( "set_HWork_Tank_3" )
      Contact( "Parametryzacja"."Time Tanks".Tank_bocking.blocing_tank3 )
      wire#w2
      Contact( "Parametryzacja"."Time Tanks".Tank_bocking.blocing_tank2 )
      wire#w3
      Contact( "Parametryzacja"."Time Tanks".Tank_bocking.blocing_tank1 )
      wire#w4
      Contact( "Parametryzacja"."Time Tanks".Tank_bocking.blocing_tank4 )
      wire#w5
      R_Coil( "Parametryzacja"."Time Tanks".Tank_bocking.blocing_tank3 )
   END_RUNG
   RUNG wire#w2
      I_Contact( "Parametryzacja"."Controls Tanks".aktywny_Zbiornik_2 )
   END_RUNG wire#w3
   RUNG wire#w3
      I_Contact( "Parametryzacja"."Controls Tanks".aktywny_Zbiornik_1 )
   END_RUNG wire#w4
   RUNG wire#w4
      I_Contact( "Parametryzacja"."Controls Tanks".aktywny_Zbiornik_4 )
   END_RUNG wire#w5
   RUNG wire#w1
      { S7_Templates := "SrcType := Word" } NE_Contact(in1 := "DB10_instance_SCADA".TrybSterowania, in2 := 2)
   END_RUNG wire#w5
   // the same network as SCL:
   IF "AlwaysFALSE" AND ((NOT "set_HWork_Tank_3" AND "Parametryzacja"."Time Tanks".Tank_bocking.blocing_tank3 AND ("Parametryzacja"."Time Tanks".Tank_bocking.blocing_tank2 OR NOT "Parametryzacja"."Controls Tanks".aktywny_Zbiornik_2) AND ("Parametryzacja"."Time Tanks".Tank_bocking.blocing_tank1 OR NOT "Parametryzacja"."Controls Tanks".aktywny_Zbiornik_1) AND ("Parametryzacja"."Time Tanks".Tank_bocking.blocing_tank4 OR NOT "Parametryzacja"."Controls Tanks".aktywny_Zbiornik_4)) OR ("DB10_instance_SCADA".TrybSterowania <> 2)) THEN
       "Parametryzacja"."Time Tanks".Tank_bocking.blocing_tank3 := FALSE;
   END_IF;
END_REGION

REGION Network 5: Zbiornik 1 ustaw jako aktywny
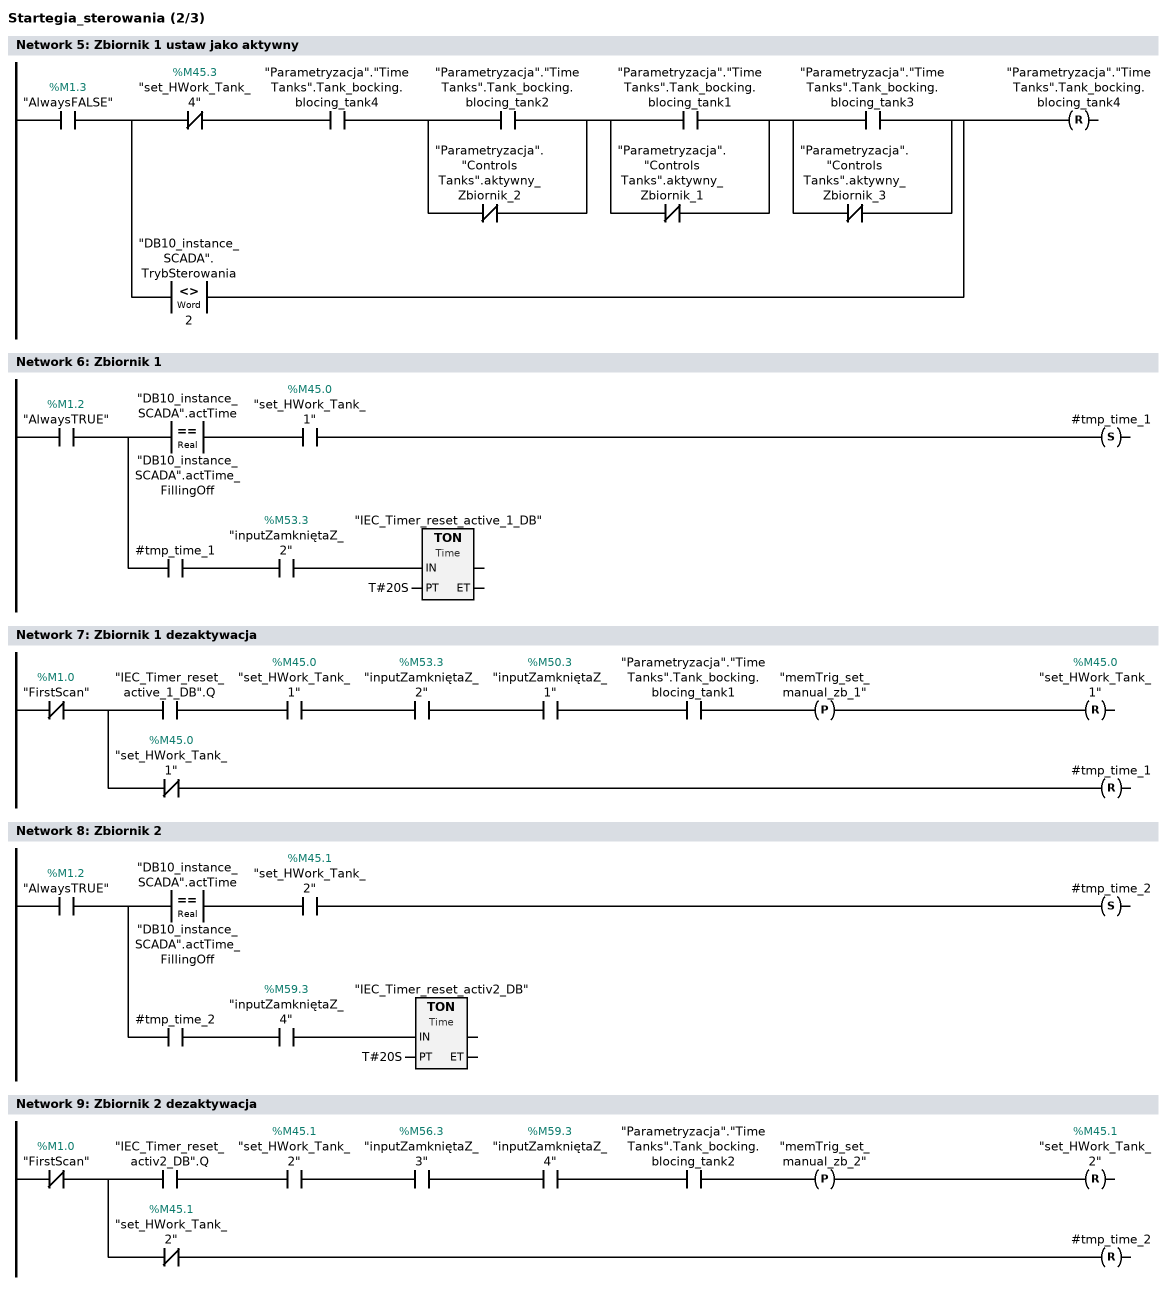
   RUNG wire#powerrail
      Contact( "AlwaysFALSE" )
      wire#w1
      I_Contact( "set_HWork_Tank_4" )
      Contact( "Parametryzacja"."Time Tanks".Tank_bocking.blocing_tank4 )
      wire#w2
      Contact( "Parametryzacja"."Time Tanks".Tank_bocking.blocing_tank2 )
      wire#w3
      Contact( "Parametryzacja"."Time Tanks".Tank_bocking.blocing_tank1 )
      wire#w4
      Contact( "Parametryzacja"."Time Tanks".Tank_bocking.blocing_tank3 )
      wire#w5
      R_Coil( "Parametryzacja"."Time Tanks".Tank_bocking.blocing_tank4 )
   END_RUNG
   RUNG wire#w2
      I_Contact( "Parametryzacja"."Controls Tanks".aktywny_Zbiornik_2 )
   END_RUNG wire#w3
   RUNG wire#w3
      I_Contact( "Parametryzacja"."Controls Tanks".aktywny_Zbiornik_1 )
   END_RUNG wire#w4
   RUNG wire#w4
      I_Contact( "Parametryzacja"."Controls Tanks".aktywny_Zbiornik_3 )
   END_RUNG wire#w5
   RUNG wire#w1
      { S7_Templates := "SrcType := Word" } NE_Contact(in1 := "DB10_instance_SCADA".TrybSterowania, in2 := 2)
   END_RUNG wire#w5
   // the same network as SCL:
   IF "AlwaysFALSE" AND ((NOT "set_HWork_Tank_4" AND "Parametryzacja"."Time Tanks".Tank_bocking.blocing_tank4 AND ("Parametryzacja"."Time Tanks".Tank_bocking.blocing_tank2 OR NOT "Parametryzacja"."Controls Tanks".aktywny_Zbiornik_2) AND ("Parametryzacja"."Time Tanks".Tank_bocking.blocing_tank1 OR NOT "Parametryzacja"."Controls Tanks".aktywny_Zbiornik_1) AND ("Parametryzacja"."Time Tanks".Tank_bocking.blocing_tank3 OR NOT "Parametryzacja"."Controls Tanks".aktywny_Zbiornik_3)) OR ("DB10_instance_SCADA".TrybSterowania <> 2)) THEN
       "Parametryzacja"."Time Tanks".Tank_bocking.blocing_tank4 := FALSE;
   END_IF;
END_REGION

REGION Network 6: Zbiornik 1
   RUNG wire#powerrail
      Contact( "AlwaysTRUE" )
      wire#w1
      { S7_Templates := "SrcType := Real" } EQ_Contact(in1 := "DB10_instance_SCADA".actTime, in2 := "DB10_instance_SCADA".actTime_FillingOff)
      Contact( "set_HWork_Tank_1" )
      S_Coil( #tmp_time_1 )
   END_RUNG
   RUNG wire#w1
      Contact( #tmp_time_1 )
      Contact( "inputZamkniętaZ_2" )
      { S7_Templates := "time_type := Time" } "IEC_Timer_reset_active_1_DB".TON(pt := T#20S, et =>)
   END_RUNG
   // the same network as SCL:
   IF "AlwaysTRUE" AND ("DB10_instance_SCADA".actTime = "DB10_instance_SCADA".actTime_FillingOff) AND "set_HWork_Tank_1" THEN
       #tmp_time_1 := TRUE;
   END_IF;
   "IEC_Timer_reset_active_1_DB".TON(IN := "AlwaysTRUE" AND #tmp_time_1 AND "inputZamkniętaZ_2", PT := T#20S);
END_REGION

REGION Network 7: Zbiornik 1 dezaktywacja
   RUNG wire#powerrail
      I_Contact( "FirstScan" )
      wire#w1
      Contact( "IEC_Timer_reset_active_1_DB".Q )
      Contact( "set_HWork_Tank_1" )
      Contact( "inputZamkniętaZ_2" )
      Contact( "inputZamkniętaZ_1" )
      Contact( "Parametryzacja"."Time Tanks".Tank_bocking.blocing_tank1 )
      P_Trig( "memTrig_set_manual_zb_1" )
      R_Coil( "set_HWork_Tank_1" )
   END_RUNG
   RUNG wire#w1
      I_Contact( "set_HWork_Tank_1" )
      R_Coil( #tmp_time_1 )
   END_RUNG
   // the same network as SCL:
   #_w1 := NOT "FirstScan" AND "IEC_Timer_reset_active_1_DB".Q AND "set_HWork_Tank_1" AND "inputZamkniętaZ_2" AND "inputZamkniętaZ_1" AND "Parametryzacja"."Time Tanks".Tank_bocking.blocing_tank1;
   #_w2 := #_w1 AND NOT "memTrig_set_manual_zb_1";   // rising edge
   "memTrig_set_manual_zb_1" := #_w1;
   IF #_w2 THEN "set_HWork_Tank_1" := FALSE; END_IF;
   IF NOT "FirstScan" AND NOT "set_HWork_Tank_1" THEN #tmp_time_1 := FALSE; END_IF;
END_REGION

REGION Network 8: Zbiornik 2
   RUNG wire#powerrail
      Contact( "AlwaysTRUE" )
      wire#w1
      { S7_Templates := "SrcType := Real" } EQ_Contact(in1 := "DB10_instance_SCADA".actTime, in2 := "DB10_instance_SCADA".actTime_FillingOff)
      Contact( "set_HWork_Tank_2" )
      S_Coil( #tmp_time_2 )
   END_RUNG
   RUNG wire#w1
      Contact( #tmp_time_2 )
      Contact( "inputZamkniętaZ_4" )
      { S7_Templates := "time_type := Time" } "IEC_Timer_reset_activ2_DB".TON(pt := T#20S, et =>)
   END_RUNG
   // the same network as SCL:
   IF "AlwaysTRUE" AND ("DB10_instance_SCADA".actTime = "DB10_instance_SCADA".actTime_FillingOff) AND "set_HWork_Tank_2" THEN
       #tmp_time_2 := TRUE;
   END_IF;
   "IEC_Timer_reset_activ2_DB".TON(IN := "AlwaysTRUE" AND #tmp_time_2 AND "inputZamkniętaZ_4", PT := T#20S);
END_REGION

REGION Network 9: Zbiornik 2 dezaktywacja
   RUNG wire#powerrail
      I_Contact( "FirstScan" )
      wire#w1
      Contact( "IEC_Timer_reset_activ2_DB".Q )
      Contact( "set_HWork_Tank_2" )
      Contact( "inputZamkniętaZ_3" )
      Contact( "inputZamkniętaZ_4" )
      Contact( "Parametryzacja"."Time Tanks".Tank_bocking.blocing_tank2 )
      P_Trig( "memTrig_set_manual_zb_2" )
      R_Coil( "set_HWork_Tank_2" )
   END_RUNG
   RUNG wire#w1
      I_Contact( "set_HWork_Tank_2" )
      R_Coil( #tmp_time_2 )
   END_RUNG
   // the same network as SCL:
   #_w1 := NOT "FirstScan" AND "IEC_Timer_reset_activ2_DB".Q AND "set_HWork_Tank_2" AND "inputZamkniętaZ_3" AND "inputZamkniętaZ_4" AND "Parametryzacja"."Time Tanks".Tank_bocking.blocing_tank2;
   #_w2 := #_w1 AND NOT "memTrig_set_manual_zb_2";   // rising edge
   "memTrig_set_manual_zb_2" := #_w1;
   IF #_w2 THEN "set_HWork_Tank_2" := FALSE; END_IF;
   IF NOT "FirstScan" AND NOT "set_HWork_Tank_2" THEN #tmp_time_2 := FALSE; END_IF;
END_REGION

REGION Network 10: Zbiornik 3
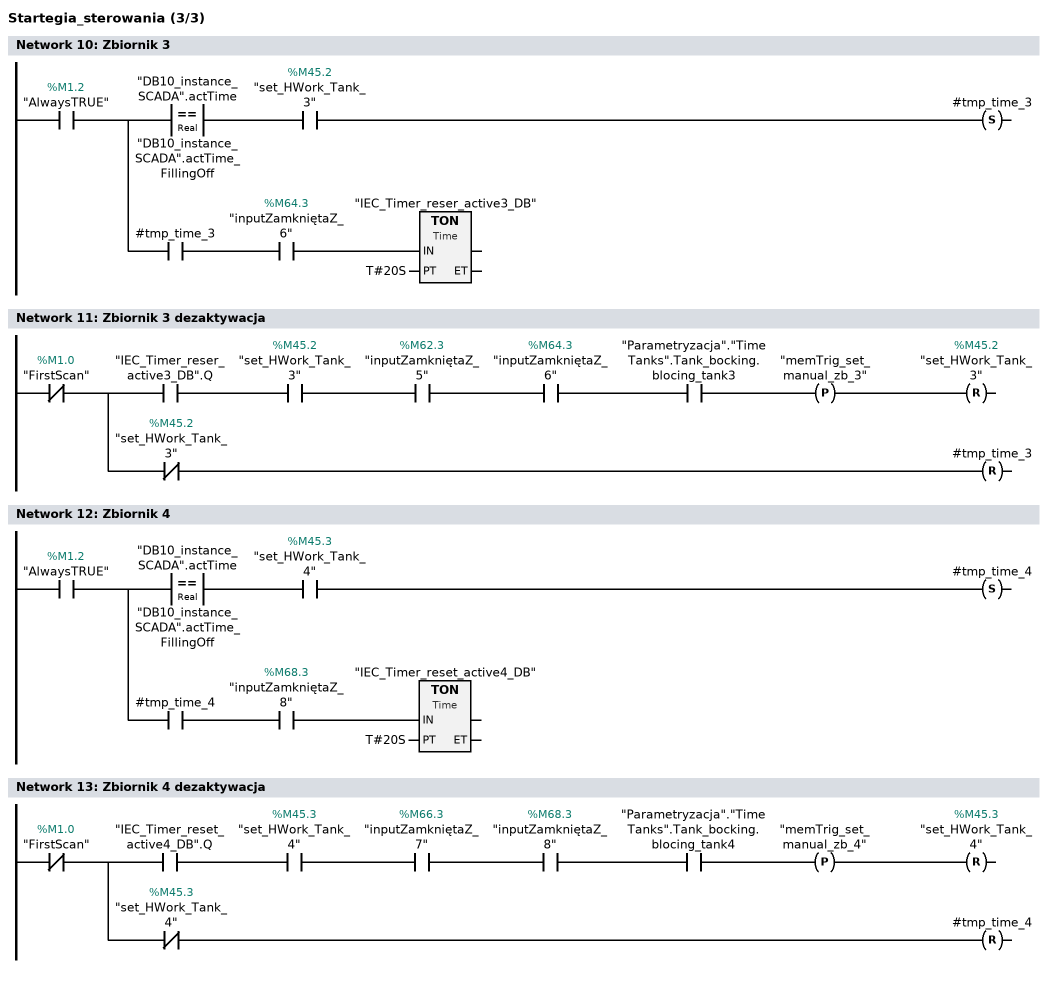
   RUNG wire#powerrail
      Contact( "AlwaysTRUE" )
      wire#w1
      { S7_Templates := "SrcType := Real" } EQ_Contact(in1 := "DB10_instance_SCADA".actTime, in2 := "DB10_instance_SCADA".actTime_FillingOff)
      Contact( "set_HWork_Tank_3" )
      S_Coil( #tmp_time_3 )
   END_RUNG
   RUNG wire#w1
      Contact( #tmp_time_3 )
      Contact( "inputZamkniętaZ_6" )
      { S7_Templates := "time_type := Time" } "IEC_Timer_reser_active3_DB".TON(pt := T#20S, et =>)
   END_RUNG
   // the same network as SCL:
   IF "AlwaysTRUE" AND ("DB10_instance_SCADA".actTime = "DB10_instance_SCADA".actTime_FillingOff) AND "set_HWork_Tank_3" THEN
       #tmp_time_3 := TRUE;
   END_IF;
   "IEC_Timer_reser_active3_DB".TON(IN := "AlwaysTRUE" AND #tmp_time_3 AND "inputZamkniętaZ_6", PT := T#20S);
END_REGION

REGION Network 11: Zbiornik 3 dezaktywacja
   RUNG wire#powerrail
      I_Contact( "FirstScan" )
      wire#w1
      Contact( "IEC_Timer_reser_active3_DB".Q )
      Contact( "set_HWork_Tank_3" )
      Contact( "inputZamkniętaZ_5" )
      Contact( "inputZamkniętaZ_6" )
      Contact( "Parametryzacja"."Time Tanks".Tank_bocking.blocing_tank3 )
      P_Trig( "memTrig_set_manual_zb_3" )
      R_Coil( "set_HWork_Tank_3" )
   END_RUNG
   RUNG wire#w1
      I_Contact( "set_HWork_Tank_3" )
      R_Coil( #tmp_time_3 )
   END_RUNG
   // the same network as SCL:
   #_w1 := NOT "FirstScan" AND "IEC_Timer_reser_active3_DB".Q AND "set_HWork_Tank_3" AND "inputZamkniętaZ_5" AND "inputZamkniętaZ_6" AND "Parametryzacja"."Time Tanks".Tank_bocking.blocing_tank3;
   #_w2 := #_w1 AND NOT "memTrig_set_manual_zb_3";   // rising edge
   "memTrig_set_manual_zb_3" := #_w1;
   IF #_w2 THEN "set_HWork_Tank_3" := FALSE; END_IF;
   IF NOT "FirstScan" AND NOT "set_HWork_Tank_3" THEN #tmp_time_3 := FALSE; END_IF;
END_REGION

REGION Network 12: Zbiornik 4
   RUNG wire#powerrail
      Contact( "AlwaysTRUE" )
      wire#w1
      { S7_Templates := "SrcType := Real" } EQ_Contact(in1 := "DB10_instance_SCADA".actTime, in2 := "DB10_instance_SCADA".actTime_FillingOff)
      Contact( "set_HWork_Tank_4" )
      S_Coil( #tmp_time_4 )
   END_RUNG
   RUNG wire#w1
      Contact( #tmp_time_4 )
      Contact( "inputZamkniętaZ_8" )
      { S7_Templates := "time_type := Time" } "IEC_Timer_reset_active4_DB".TON(pt := T#20S, et =>)
   END_RUNG
   // the same network as SCL:
   IF "AlwaysTRUE" AND ("DB10_instance_SCADA".actTime = "DB10_instance_SCADA".actTime_FillingOff) AND "set_HWork_Tank_4" THEN
       #tmp_time_4 := TRUE;
   END_IF;
   "IEC_Timer_reset_active4_DB".TON(IN := "AlwaysTRUE" AND #tmp_time_4 AND "inputZamkniętaZ_8", PT := T#20S);
END_REGION

REGION Network 13: Zbiornik 4 dezaktywacja
   RUNG wire#powerrail
      I_Contact( "FirstScan" )
      wire#w1
      Contact( "IEC_Timer_reset_active4_DB".Q )
      Contact( "set_HWork_Tank_4" )
      Contact( "inputZamkniętaZ_7" )
      Contact( "inputZamkniętaZ_8" )
      Contact( "Parametryzacja"."Time Tanks".Tank_bocking.blocing_tank4 )
      P_Trig( "memTrig_set_manual_zb_4" )
      R_Coil( "set_HWork_Tank_4" )
   END_RUNG
   RUNG wire#w1
      I_Contact( "set_HWork_Tank_4" )
      R_Coil( #tmp_time_4 )
   END_RUNG
   // the same network as SCL:
   #_w1 := NOT "FirstScan" AND "IEC_Timer_reset_active4_DB".Q AND "set_HWork_Tank_4" AND "inputZamkniętaZ_7" AND "inputZamkniętaZ_8" AND "Parametryzacja"."Time Tanks".Tank_bocking.blocing_tank4;
   #_w2 := #_w1 AND NOT "memTrig_set_manual_zb_4";   // rising edge
   "memTrig_set_manual_zb_4" := #_w1;
   IF #_w2 THEN "set_HWork_Tank_4" := FALSE; END_IF;
   IF NOT "FirstScan" AND NOT "set_HWork_Tank_4" THEN #tmp_time_4 := FALSE; END_IF;
END_REGION
END_FUNCTION_BLOCK

FUNCTION_BLOCK "godzinyPracy"   // FB19, LAD
{ S7_Optimized_Access := 'TRUE' }
AUTHOR : RTecmer
FAMILY : XMHour
VERSION : 0.1
// Licznik czasu pracy
// stored: AutoNumber true, IsIECCheckEnabled false, IsRetainMemResEnabled false, MemoryReserve 500, SetENOAutomatically false, UDAEnableTagReadback false
   VAR_INPUT
      Run_Device : Bool;
   END_VAR
   VAR_OUTPUT
      MW_hour : DWord;
      Sum_hour_sek : Real;   // Licznik sumator godzin i sekund na potrzeby wyznaczania dumchawy do pracy
   END_VAR
   VAR_IN_OUT
      Data_sek : Int;
      Reset { ExternalAccessible := 'False'; ExternalVisible := 'False'; ExternalWritable := 'False'} : Bool;
      Data_hour : DWord;
      Edge_Hz { ExternalAccessible := 'False'; ExternalVisible := 'False'; ExternalWritable := 'False'} : Bool;
   END_VAR
   VAR
      sek_real { ExternalAccessible := 'False'; ExternalVisible := 'False'; ExternalWritable := 'False'} : Real;   // pomocnicza konwerski sekund
      actSekReal { ExternalAccessible := 'False'; ExternalVisible := 'False'; ExternalWritable := 'False'} : Real;   // aktualne sekundy po konwersji
      hour_sek { ExternalAccessible := 'False'; ExternalVisible := 'False'; ExternalWritable := 'False'} : Real;
   END_VAR
   VAR_TEMP   // added for the SCL form of the ladder/FBD networks
      _w1 : Bool;
      _w2 : Bool;
   END_VAR
BEGIN

REGION Network 1
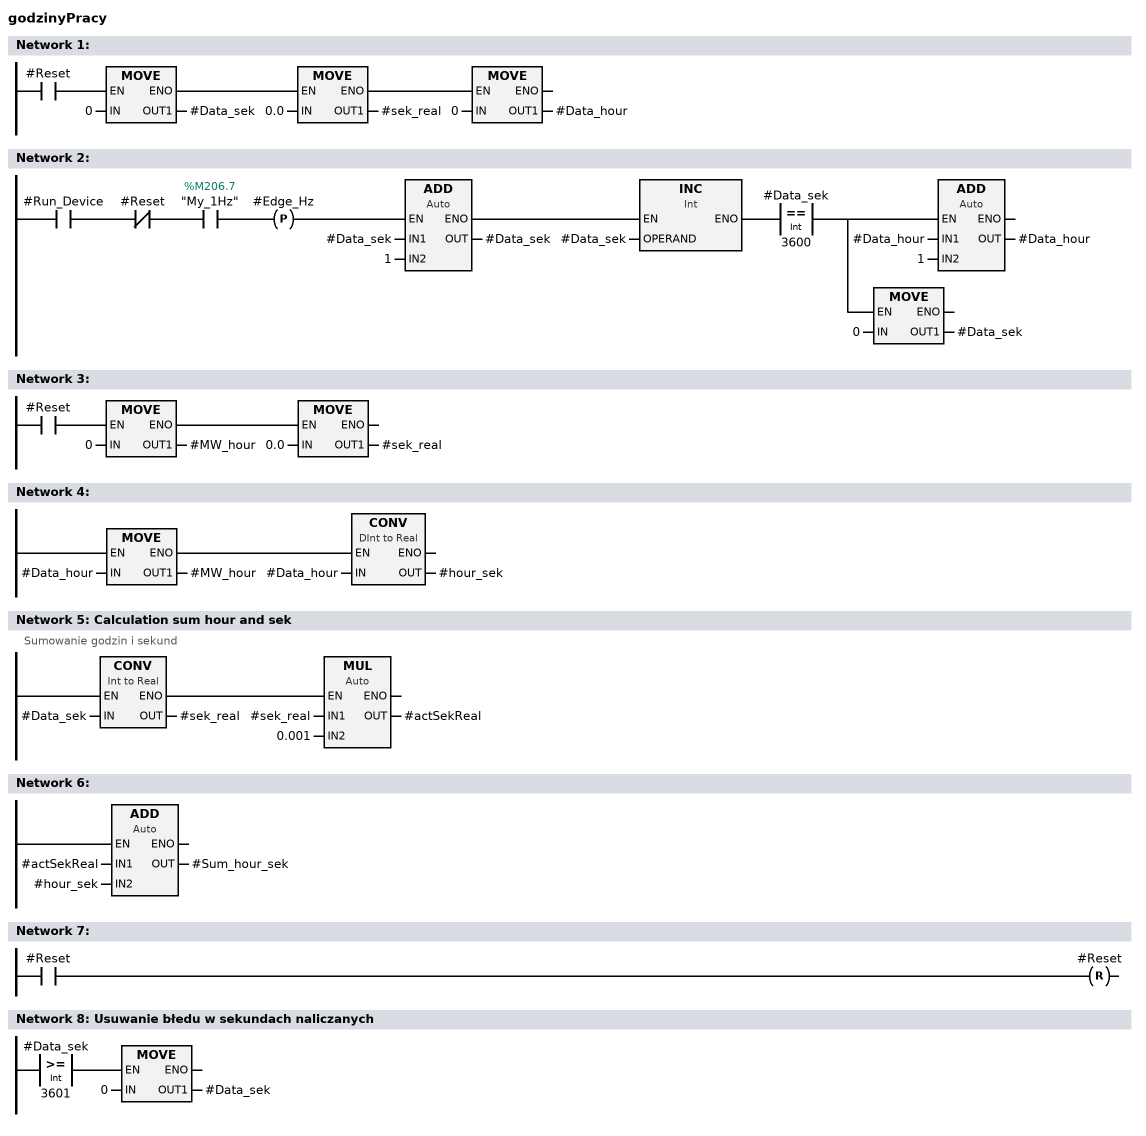
   RUNG wire#powerrail
      Contact( #Reset )
      { S7_GenerateENO := "TRUE" } Move(in := 0, out1 => #Data_sek)
      { S7_GenerateENO := "TRUE" } Move(in := 0.0, out1 => #sek_real)
      { S7_GenerateENO := "TRUE" } Move(in := 0, out1 => #Data_hour)
   END_RUNG
   // the same network as SCL:
   // ENO of a box is taken as its EN; it also drops when the box reports an error
   IF #Reset THEN
       #Data_sek := 0;
       #sek_real := 0.0;
       #Data_hour := 0;
   END_IF;
END_REGION

REGION Network 2
   RUNG wire#powerrail
      Contact( #Run_Device )
      I_Contact( #Reset )
      Contact( "My_1Hz" )
      P_Trig( #Edge_Hz )
      { S7_GenerateENO := "TRUE" } Add(in1 := #Data_sek, in2 := 1, out => #Data_sek)
      { S7_Templates := "DestType := Int"; S7_GenerateENO := "TRUE" } Inc( #Data_sek )
      { S7_Templates := "SrcType := Int" } EQ_Contact(in1 := #Data_sek, in2 := 3600)
      wire#w1
      { S7_GenerateENO := "TRUE" } Add(in1 := #Data_hour, in2 := 1, out => #Data_hour)
   END_RUNG
   RUNG wire#w1
      { S7_GenerateENO := "TRUE" } Move(in := 0, out1 => #Data_sek)
   END_RUNG
   // the same network as SCL:
   // ENO of a box is taken as its EN; it also drops when the box reports an error
   #_w1 := #Run_Device AND NOT #Reset AND "My_1Hz";
   #_w2 := #_w1 AND NOT #Edge_Hz;   // rising edge
   #Edge_Hz := #_w1;
   IF #_w2 THEN
       #Data_sek := #Data_sek + 1;
       #Data_sek := #Data_sek + 1;
   END_IF;
   IF #_w2 AND (#Data_sek = 3600) THEN
       #Data_hour := #Data_hour + 1;
       #Data_sek := 0;
   END_IF;
END_REGION

REGION Network 3
   RUNG wire#powerrail
      Contact( #Reset )
      { S7_GenerateENO := "TRUE" } Move(in := 0, out1 => #MW_hour)
      { S7_GenerateENO := "TRUE" } Move(in := 0.0, out1 => #sek_real)
   END_RUNG
   // the same network as SCL:
   // ENO of a box is taken as its EN; it also drops when the box reports an error
   IF #Reset THEN
       #MW_hour := 0;
       #sek_real := 0.0;
   END_IF;
END_REGION

REGION Network 4
   RUNG wire#powerrail
      { S7_GenerateENO := "TRUE" } Move(in := #Data_hour, out1 => #MW_hour)
      { S7_Templates := "[SrcType := DInt, DestType := Real]" } Convert(in := #Data_hour, out => #hour_sek)
   END_RUNG
   // the same network as SCL:
   // ENO of a box is taken as its EN; it also drops when the box reports an error
   #MW_hour := #Data_hour;
   #hour_sek := DINT_TO_REAL(#Data_hour);
END_REGION

REGION Network 5: Calculation sum hour and sek
   // Sumowanie godzin i sekund
   RUNG wire#powerrail
      { S7_Templates := "[SrcType := Int, DestType := Real]" } Convert(in := #Data_sek, out => #sek_real)
      Mul(in1 := #sek_real, in2 := 0.001, out => #actSekReal)
   END_RUNG
   // the same network as SCL:
   #sek_real := INT_TO_REAL(#Data_sek);
   #actSekReal := #sek_real * 0.001;
END_REGION

REGION Network 6
   RUNG wire#powerrail
      Add(in1 := #actSekReal, in2 := #hour_sek, out => #Sum_hour_sek)
   END_RUNG
   // the same network as SCL:
   #Sum_hour_sek := #actSekReal + #hour_sek;
END_REGION

REGION Network 7
   RUNG wire#powerrail
      Contact( #Reset )
      R_Coil( #Reset )
   END_RUNG
   // the same network as SCL:
   IF #Reset THEN #Reset := FALSE; END_IF;
END_REGION

REGION Network 8: Usuwanie błedu w sekundach naliczanych
   RUNG wire#powerrail
      { S7_Templates := "SrcType := Int" } GE_Contact(in1 := #Data_sek, in2 := 3601)
      { S7_GenerateENO := "TRUE" } Move(in := 0, out1 => #Data_sek)
   END_RUNG
   // the same network as SCL:
   IF #Data_sek >= 3601 THEN #Data_sek := 0; END_IF;
END_REGION
END_FUNCTION_BLOCK

FUNCTION "Sterowanie_Zbiornik" : Void   // FC26, LAD
TITLE = Napełnianie i opróżnianie
{ S7_Optimized_Access := 'TRUE' }
AUTHOR : rtecmer
VERSION : 0.1
// Funkcja steruje napędami napełniania i opróżniania w cyklu od zegara czasu jak i od pomiaru poziomu. Poziom jest sygnałem nadrzędnym. Jeśli napełnienie uzyskano przed czasem to napełnianie jest kończone z osiągnięciem poziomu max. Podczas oróżniania jeśli osiągnięto poziom min to opróżnianie zbiorniak jest zakończone.
// Granica końca minimum to 100cm ponad tę wartość nastąpi dopiero skasowanie sygnału poziom MIN
// Spadku poziomu poniżej 250cm pozwala na scasowanie sygnału poziom MAX
// stored: AutoNumber true, IsIECCheckEnabled false, SetENOAutomatically false, UDAEnableTagReadback false
   VAR_INPUT
      actLevel : Real;   // pozim w zbiorniku
      maxLevel : Real;   // poziom napełnienia
      minLevel : Real;   // poziom opróżnienia
      actTime : Real;   // czas aktualny
      actTime_FillingOn : Real;   // godzina start napełnianie
      actTime_FillingOff : Real;   // godzina stop napełnianie
      actTime_EmptyingOn : Real;   // godzina start przetłaczanie
      actTime_EmptyingOff : Real;   // godzina stop przetłaczanie
      isOpen_filling : Bool;   // potwierdzenie otwarcia napełniającej zasuwy
      isOpen_emptying : Bool;   // potwierdzenie otwarcia spustowej zasuwy
      isClose_filling : Bool;   // potwierdzenie zamknięcia napełniającej zasuwy
      isClose_emptying : Bool;   // potwierdzenie zamknięcia spustowej zasuwy
      isReady_filling : Bool;   // sygnał gotowości zasuwa napełnianie
      isReadyt_emptying : Bool;   // sygnał gotowości zasuwa spustowa
      activTank : Bool;   // zbiornik aktywny
      isAut_Valve_Filling : Bool;   // tryb pracy automat zasuwa napełnianie
      isAut_Valve_Empting : Bool;   // tryb pracy automat zasuwa spustowa
      is_min_Float : Bool;   // sygnał minimum z płyawaka
      is_max_Float : Bool;   // sygnał max z płyawaka
      isAlarmNinimum_barB5 : Bool;   // alarm niskie ciśnienie magistrala
      resetAlarmMinimum_barB5 : Bool;   // koniec alarm niskie ciśnienie magistral
      setTank_Work_daily : Bool;   // tryb pracy dobowy aktywny
      setTank_Work_selective : Bool;   // tryb pracy selektywny - jeden zbiornik aktywny
      setControl_alarm_B5 : Bool;   // sygnał uruchomienie awaryjnego otwarcie zbiornika na dosilanie
      set_HWork_tank : Bool;   // ustawia aktywny zbiornik do pracy w trybie selektywnym
   END_VAR
   VAR_OUTPUT
      setSVMO_Z_Wlot : Bool;   // bit otwierania w trybie automat
      setSVMC_Z_Wlot : Bool;   // bit zamykania w trybie automat
      setSVMO_Z_Spust : Bool;   // bit otwierania w trybie automat
      setSVMC_Z_Spust : Bool;   // bit zamykania w trybie automat
      infoFiling_to_HMI : Bool;   // bit informacji wejściu w tryb napełniania
   END_VAR
   VAR_IN_OUT
      isFilling : Bool;   // bit aktywacji napełninia
      isEptying : Bool;   // bit aktywacji przetłaczania
      memRisingLevel_min : Bool;   // pamięc zbocza osiągniecia poziomu minimum w zbiorniku
      memRisingLevel_max : Bool;   // pamięc zbocza osiągniecia poziomu max w zbiorniku
      isLevelMax : Bool;   // poziom max
      isLevelMin : Bool;   // poziom min
      blok_tank : Bool;   // bit blokowania zbiornika w sekwencji
   END_VAR
   VAR_TEMP
      correction_max : Real;   // współczynnik korekty dla zachowania histerezy przy wahaniu poziomu w zbiorniku
      correction_min : Real;   // współczynnik korekty dla zachowania histerezy przy wahaniu poziomu w zbiorniku
      filling_time : Real;   // wyliczony czas napełniania na dobę
      filing_time_X : Bool;   // bit logika gdy napełnianie przed 00:00
      filing_time_Y : Bool;   // bit logika gdy napełnianie po 00:01
      epting_time_X : Bool;   // bit logika gdy napełnianie po 00:01
   END_VAR
   VAR_TEMP   // added for the SCL form of the ladder/FBD networks
      _w1 : Bool;
      _w2 : Bool;
   END_VAR
BEGIN

REGION Network 1 (SCL): wyliczenie korekty dla stabilności sygału min i max
   #correction_max := (#maxLevel - 30);
   #correction_min := (#minLevel + 20);
END_REGION

REGION Network 2: znacznik poziom max
   // przechwycenie poziomu max
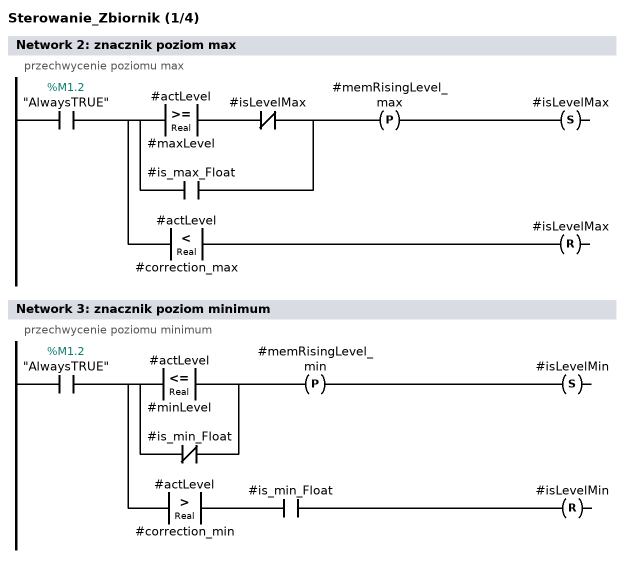
   RUNG wire#powerrail
      Contact( "AlwaysTRUE" )
      wire#w1
      { S7_Templates := "SrcType := Real" } GE_Contact(in1 := #actLevel, in2 := #maxLevel)
      I_Contact( #isLevelMax )
      wire#w2
      P_Trig( #memRisingLevel_max )
      S_Coil( #isLevelMax )
   END_RUNG
   RUNG wire#w1
      Contact( #is_max_Float )
   END_RUNG wire#w2
   RUNG wire#w1
      { S7_Templates := "SrcType := Real" } LT_Contact(in1 := #actLevel, in2 := #correction_max)
      R_Coil( #isLevelMax )
   END_RUNG
   // the same network as SCL:
   #_w1 := "AlwaysTRUE" AND (((#actLevel >= #maxLevel) AND NOT #isLevelMax) OR #is_max_Float);
   #_w2 := #_w1 AND NOT #memRisingLevel_max;   // rising edge
   #memRisingLevel_max := #_w1;
   IF #_w2 THEN #isLevelMax := TRUE; END_IF;
   IF "AlwaysTRUE" AND (#actLevel < #correction_max) THEN #isLevelMax := FALSE; END_IF;
END_REGION

REGION Network 3: znacznik poziom minimum
   // przechwycenie poziomu minimum
   RUNG wire#powerrail
      Contact( "AlwaysTRUE" )
      wire#w1
      { S7_Templates := "SrcType := Real" } LE_Contact(in1 := #actLevel, in2 := #minLevel)
      wire#w2
      P_Trig( #memRisingLevel_min )
      S_Coil( #isLevelMin )
   END_RUNG
   RUNG wire#w1
      I_Contact( #is_min_Float )
   END_RUNG wire#w2
   RUNG wire#w1
      { S7_Templates := "SrcType := Real" } GT_Contact(in1 := #actLevel, in2 := #correction_min)
      Contact( #is_min_Float )
      R_Coil( #isLevelMin )
   END_RUNG
   // the same network as SCL:
   #_w1 := "AlwaysTRUE" AND ((#actLevel <= #minLevel) OR NOT #is_min_Float);
   #_w2 := #_w1 AND NOT #memRisingLevel_min;   // rising edge
   #memRisingLevel_min := #_w1;
   IF #_w2 THEN #isLevelMin := TRUE; END_IF;
   IF "AlwaysTRUE" AND (#actLevel > #correction_min) AND #is_min_Float THEN #isLevelMin := FALSE; END_IF;
END_REGION

REGION Network 4 (SCL): wyliczony czas napełniania na dobę i ustawoanie bitu kontroli pracy w dobie
   // #filing_time_X  - bit ustawiany w przypadku gdy w przedziale pracy wystąpi przejście przez  godzinę 00:00
   IF #actTime_FillingOn > #actTime_FillingOff THEN
     // odejmnij od wiekszej mniejszą
     #filling_time := (#actTime_FillingOn - #actTime_FillingOff);
     IF #actTime >=  #actTime_FillingOn THEN
       // jeśli czas rozpoczęcia napełniania to ustaw bit
       #filing_time_X := TRUE;
       ;
     ELSE
       // w innym wypadku kasuj bit
       #filing_time_X := False;
       ;
     END_IF;

     #filing_time_Y := FALSE;
   ELSE
     #filling_time := (#actTime_FillingOff - #actTime_FillingOn);
     #filing_time_X := False;
     #filing_time_Y := TRUE;
     ;
   END_IF;
END_REGION

REGION Network 5: bit aktywacji napełninia
   // aktywacja, deaktywacja bitu rocedury napełniania
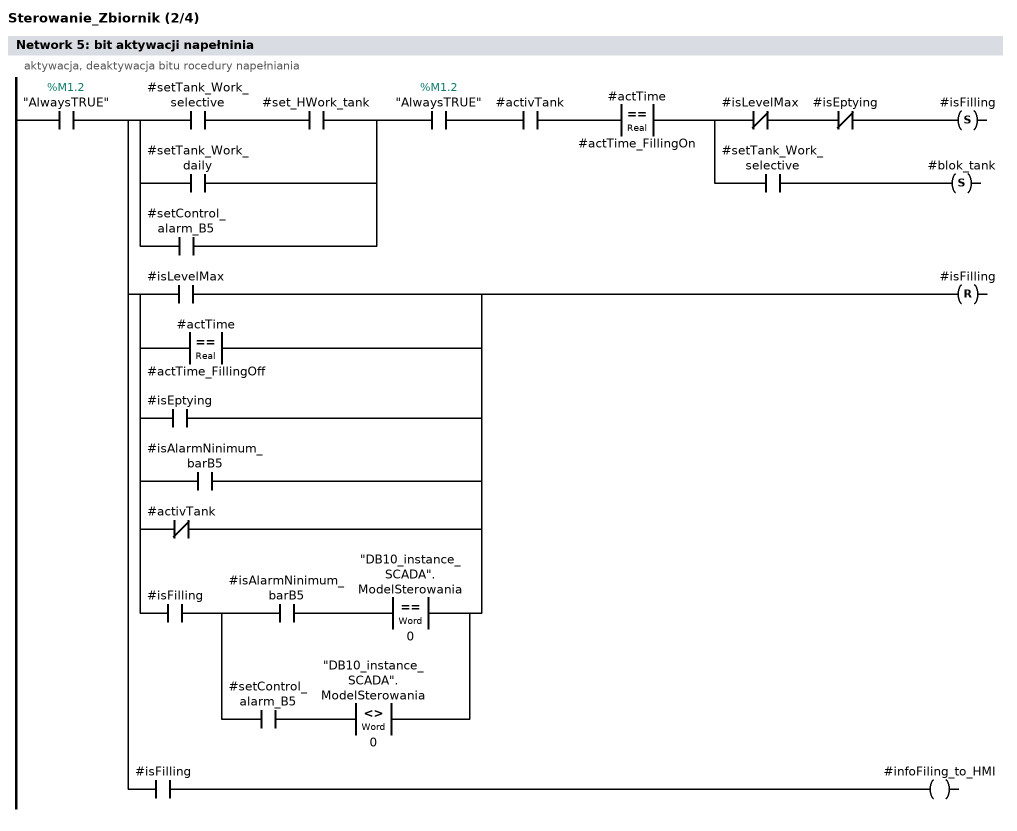
   RUNG wire#powerrail
      Contact( "AlwaysTRUE" )
      wire#w1
      Contact( #setTank_Work_selective )
      Contact( #set_HWork_tank )
      wire#w2
      Contact( "AlwaysTRUE" )
      Contact( #activTank )
      { S7_Templates := "SrcType := Real" } EQ_Contact(in1 := #actTime, in2 := #actTime_FillingOn)
      wire#w3
      I_Contact( #isLevelMax )
      I_Contact( #isEptying )
      S_Coil( #isFilling )
   END_RUNG
   RUNG wire#w1
      Contact( #setTank_Work_daily )
   END_RUNG wire#w2
   RUNG wire#w1
      Contact( #setControl_alarm_B5 )
   END_RUNG wire#w2
   RUNG wire#w3
      Contact( #setTank_Work_selective )
      S_Coil( #blok_tank )
   END_RUNG
   RUNG wire#w1
      Contact( #isLevelMax )
      wire#w4
      R_Coil( #isFilling )
   END_RUNG
   RUNG wire#w1
      { S7_Templates := "SrcType := Real" } EQ_Contact(in1 := #actTime, in2 := #actTime_FillingOff)
   END_RUNG wire#w4
   RUNG wire#w1
      Contact( #isEptying )
   END_RUNG wire#w4
   RUNG wire#w1
      Contact( #isAlarmNinimum_barB5 )
   END_RUNG wire#w4
   RUNG wire#w1
      I_Contact( #activTank )
   END_RUNG wire#w4
   RUNG wire#w1
      Contact( #isFilling )
      wire#w5
      Contact( #isAlarmNinimum_barB5 )
      { S7_Templates := "SrcType := Word" } EQ_Contact(in1 := "DB10_instance_SCADA".ModelSterowania, in2 := 0)
   END_RUNG wire#w4
   RUNG wire#w5
      Contact( #setControl_alarm_B5 )
      { S7_Templates := "SrcType := Word" } NE_Contact(in1 := "DB10_instance_SCADA".ModelSterowania, in2 := 0)
   END_RUNG wire#w4
   RUNG wire#w1
      Contact( #isFilling )
      Coil( #infoFiling_to_HMI )
   END_RUNG
   // the same network as SCL:
   #_w1 := "AlwaysTRUE" AND ((#setTank_Work_selective AND #set_HWork_tank) OR #setTank_Work_daily OR #setControl_alarm_B5) AND "AlwaysTRUE" AND #activTank AND (#actTime = #actTime_FillingOn);
   IF #_w1 AND NOT #isLevelMax AND NOT #isEptying THEN #isFilling := TRUE; END_IF;
   IF #_w1 AND #setTank_Work_selective THEN #blok_tank := TRUE; END_IF;
   IF "AlwaysTRUE" AND (#isLevelMax OR (#actTime = #actTime_FillingOff) OR #isEptying OR #isAlarmNinimum_barB5 OR NOT #activTank OR (#isFilling AND ((#isAlarmNinimum_barB5 AND ("DB10_instance_SCADA".ModelSterowania = 0)) OR (#setControl_alarm_B5 AND ("DB10_instance_SCADA".ModelSterowania <> 0))))) THEN
       #isFilling := FALSE;
   END_IF;
   #infoFiling_to_HMI := "AlwaysTRUE" AND #isFilling;
END_REGION

REGION Network 6 (SCL): ustawoanie bitu kontroli pracy w dobie
   // epting_time_X  - bit ustawiany w przypadku gdy w przedziale pracy wystąpi przejście przez  godzinę 00:00
   IF #actTime_EmptyingOn > #actTime_EmptyingOff THEN

     IF #actTime >=  #actTime_EmptyingOn THEN
       // jeśli czas rozpoczęcia napełniania to ustaw bit
       #epting_time_X := TRUE;
       ;
     ELSE
       // w innym wypadku kasuj bit
       #epting_time_X := False;
       ;
     END_IF;

   ELSE

     #epting_time_X := False;

     ;
   END_IF;
END_REGION

REGION Network 7: bit aktywacji przetłaczania
   // aktywacja/ deaktywacja bitu pracy pompowni (przetłaczanie)
   // musi zakonczyć się napełnianie, jeśli wyłaczysz z trybu automat to reset znacznika przetłaczanie
   // 
   // #epting_time_X - usunąłem na testy
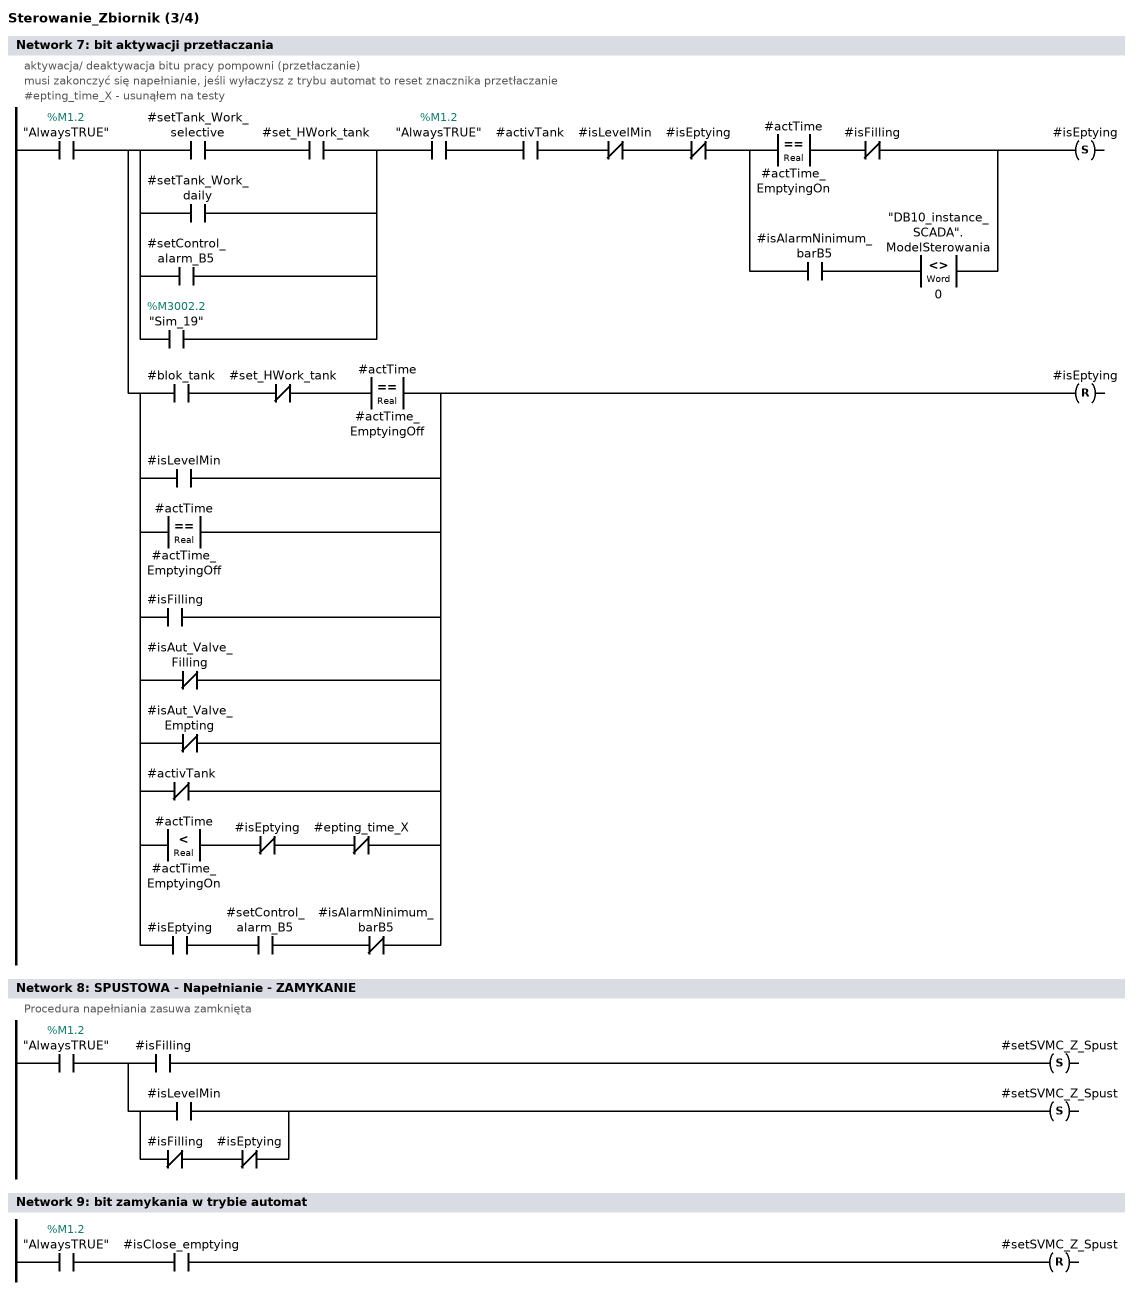
   RUNG wire#powerrail
      Contact( "AlwaysTRUE" )
      wire#w1
      Contact( #setTank_Work_selective )
      Contact( #set_HWork_tank )
      wire#w2
      Contact( "AlwaysTRUE" )
      Contact( #activTank )
      I_Contact( #isLevelMin )
      I_Contact( #isEptying )
      wire#w3
      { S7_Templates := "SrcType := Real" } EQ_Contact(in1 := #actTime, in2 := #actTime_EmptyingOn)
      I_Contact( #isFilling )
      wire#w4
      S_Coil( #isEptying )
   END_RUNG
   RUNG wire#w1
      Contact( #setTank_Work_daily )
   END_RUNG wire#w2
   RUNG wire#w1
      Contact( #setControl_alarm_B5 )
   END_RUNG wire#w2
   RUNG wire#w1
      Contact( "Sim_19" )
   END_RUNG wire#w2
   RUNG wire#w3
      Contact( #isAlarmNinimum_barB5 )
      { S7_Templates := "SrcType := Word" } NE_Contact(in1 := "DB10_instance_SCADA".ModelSterowania, in2 := 0)
   END_RUNG wire#w4
   RUNG wire#w1
      Contact( #blok_tank )
      I_Contact( #set_HWork_tank )
      { S7_Templates := "SrcType := Real" } EQ_Contact(in1 := #actTime, in2 := #actTime_EmptyingOff)
      wire#w5
      R_Coil( #isEptying )
   END_RUNG
   RUNG wire#w1
      Contact( #isLevelMin )
   END_RUNG wire#w5
   RUNG wire#w1
      { S7_Templates := "SrcType := Real" } EQ_Contact(in1 := #actTime, in2 := #actTime_EmptyingOff)
   END_RUNG wire#w5
   RUNG wire#w1
      Contact( #isFilling )
   END_RUNG wire#w5
   RUNG wire#w1
      I_Contact( #isAut_Valve_Filling )
   END_RUNG wire#w5
   RUNG wire#w1
      I_Contact( #isAut_Valve_Empting )
   END_RUNG wire#w5
   RUNG wire#w1
      I_Contact( #activTank )
   END_RUNG wire#w5
   RUNG wire#w1
      { S7_Templates := "SrcType := Real" } LT_Contact(in1 := #actTime, in2 := #actTime_EmptyingOn)
      I_Contact( #isEptying )
      I_Contact( #epting_time_X )
   END_RUNG wire#w5
   RUNG wire#w1
      Contact( #isEptying )
      Contact( #setControl_alarm_B5 )
      I_Contact( #isAlarmNinimum_barB5 )
   END_RUNG wire#w5
   // the same network as SCL:
   IF "AlwaysTRUE" AND ((#setTank_Work_selective AND #set_HWork_tank) OR #setTank_Work_daily OR #setControl_alarm_B5 OR "Sim_19") AND "AlwaysTRUE" AND #activTank AND NOT #isLevelMin AND NOT #isEptying AND (((#actTime = #actTime_EmptyingOn) AND NOT #isFilling) OR (#isAlarmNinimum_barB5 AND ("DB10_instance_SCADA".ModelSterowania <> 0))) THEN
       #isEptying := TRUE;
   END_IF;
   IF "AlwaysTRUE" AND ((#blok_tank AND NOT #set_HWork_tank AND (#actTime = #actTime_EmptyingOff)) OR #isLevelMin OR (#actTime = #actTime_EmptyingOff) OR #isFilling OR NOT #isAut_Valve_Filling OR NOT #isAut_Valve_Empting OR NOT #activTank OR ((#actTime < #actTime_EmptyingOn) AND NOT #isEptying AND NOT #epting_time_X) OR (#isEptying AND #setControl_alarm_B5 AND NOT #isAlarmNinimum_barB5)) THEN
       #isEptying := FALSE;
   END_IF;
END_REGION

REGION Network 8: SPUSTOWA - Napełnianie - ZAMYKANIE
   // Procedura napełniania zasuwa zamknięta
   RUNG wire#powerrail
      Contact( "AlwaysTRUE" )
      wire#w1
      Contact( #isFilling )
      S_Coil( #setSVMC_Z_Spust )
   END_RUNG
   RUNG wire#w1
      Contact( #isLevelMin )
      wire#w2
      S_Coil( #setSVMC_Z_Spust )
   END_RUNG
   RUNG wire#w1
      I_Contact( #isFilling )
      I_Contact( #isEptying )
   END_RUNG wire#w2
   // the same network as SCL:
   IF "AlwaysTRUE" AND #isFilling THEN #setSVMC_Z_Spust := TRUE; END_IF;
   IF "AlwaysTRUE" AND (#isLevelMin OR (NOT #isFilling AND NOT #isEptying)) THEN
       #setSVMC_Z_Spust := TRUE;
   END_IF;
END_REGION

REGION Network 9: bit zamykania w trybie automat
   RUNG wire#powerrail
      Contact( "AlwaysTRUE" )
      Contact( #isClose_emptying )
      R_Coil( #setSVMC_Z_Spust )
   END_RUNG
   // the same network as SCL:
   IF "AlwaysTRUE" AND #isClose_emptying THEN #setSVMC_Z_Spust := FALSE; END_IF;
END_REGION

REGION Network 10: bit otwierania w trybie automat - OTWIERANIE
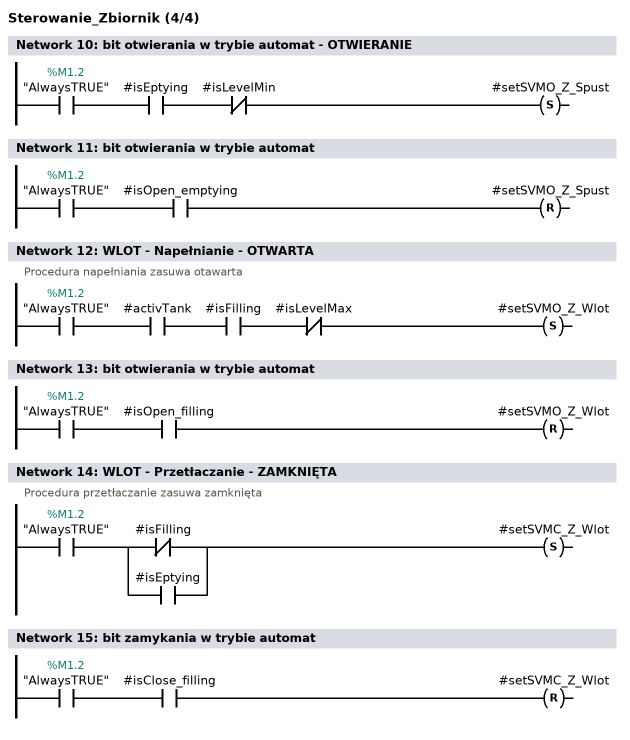
   RUNG wire#powerrail
      Contact( "AlwaysTRUE" )
      Contact( #isEptying )
      I_Contact( #isLevelMin )
      S_Coil( #setSVMO_Z_Spust )
   END_RUNG
   // the same network as SCL:
   IF "AlwaysTRUE" AND #isEptying AND NOT #isLevelMin THEN #setSVMO_Z_Spust := TRUE; END_IF;
END_REGION

REGION Network 11: bit otwierania w trybie automat
   RUNG wire#powerrail
      Contact( "AlwaysTRUE" )
      Contact( #isOpen_emptying )
      R_Coil( #setSVMO_Z_Spust )
   END_RUNG
   // the same network as SCL:
   IF "AlwaysTRUE" AND #isOpen_emptying THEN #setSVMO_Z_Spust := FALSE; END_IF;
END_REGION

REGION Network 12: WLOT - Napełnianie - OTWARTA
   // Procedura napełniania zasuwa otawarta
   RUNG wire#powerrail
      Contact( "AlwaysTRUE" )
      Contact( #activTank )
      Contact( #isFilling )
      I_Contact( #isLevelMax )
      S_Coil( #setSVMO_Z_Wlot )
   END_RUNG
   // the same network as SCL:
   IF "AlwaysTRUE" AND #activTank AND #isFilling AND NOT #isLevelMax THEN #setSVMO_Z_Wlot := TRUE; END_IF;
END_REGION

REGION Network 13: bit otwierania w trybie automat
   RUNG wire#powerrail
      Contact( "AlwaysTRUE" )
      Contact( #isOpen_filling )
      R_Coil( #setSVMO_Z_Wlot )
   END_RUNG
   // the same network as SCL:
   IF "AlwaysTRUE" AND #isOpen_filling THEN #setSVMO_Z_Wlot := FALSE; END_IF;
END_REGION

REGION Network 14: WLOT - Przetłaczanie - ZAMKNIĘTA
   // Procedura przetłaczanie zasuwa zamknięta
   RUNG wire#powerrail
      Contact( "AlwaysTRUE" )
      wire#w1
      I_Contact( #isFilling )
      wire#w2
      S_Coil( #setSVMC_Z_Wlot )
   END_RUNG
   RUNG wire#w1
      Contact( #isEptying )
   END_RUNG wire#w2
   // the same network as SCL:
   IF "AlwaysTRUE" AND (NOT #isFilling OR #isEptying) THEN #setSVMC_Z_Wlot := TRUE; END_IF;
END_REGION

REGION Network 15: bit zamykania w trybie automat
   RUNG wire#powerrail
      Contact( "AlwaysTRUE" )
      Contact( #isClose_filling )
      R_Coil( #setSVMC_Z_Wlot )
   END_RUNG
   // the same network as SCL:
   IF "AlwaysTRUE" AND #isClose_filling THEN #setSVMC_Z_Wlot := FALSE; END_IF;
END_REGION
END_FUNCTION

FUNCTION "Sterowania _Zasuwa_Z9" : Void
TITLE = Sterowanie zasuwą Z9 odpływu ze zbiorników
{ S7_Optimized_Access := 'TRUE' }
AUTHOR : rtecmr
VERSION : 0.1
//Otwieranie zasuwy w cyklu przetłaczania, dosilania. PLC Pompownia na podstawie statusu zasuwy Z9 i bitu informującego o otwarciu rozoczyna procedurę przetłaczania lub dosilania
   VAR_INPUT 
      isGotowość : Bool;   // bit gotowości
      isAuto : Bool;   // bit trybu autoamt
      isOpen : Bool;   // potwierdzenia otwarta
      isClose : Bool;   // potwierdzenia zamknieta
      isPumping : Bool;   // bit wybrano tryb przetłaczania
      isRecharging : Bool;   // bit wybrano tryb dosilania
      isAutPumping : Bool;   // bit wybrano tryb automatycznego sterowania pompownią tryb mieszany dosilania-przetłaczanie
      isREM : Bool;   // bit przełacznik trybu pracy załaczony
   END_VAR

   VAR_OUTPUT 
      setSVMC : Bool;   // bit rozkazu zamyknij w automacie
      setSVMO : Bool;   // bit rozkazu otwórz w automacie
   END_VAR


BEGIN
	(*
	//=============================================================================
	//(JZWiK S.A Radosław Tecmer)
	//(c)Copyright (2022) All Rights Reserved
	//-----------------------------------------------------------------------------
	//Testowane z:   (system docelowy z  FW 4.4)
	//Pakiet inżynierski:   TIA Portal (V16 Update 5)
	//Ograniczenia:  ( - )
	//Wymagania:  (minimalne S7-1200 CPU 1215C FW 4.2 .)
	//Funkcjonalnośc: (Sterowanie zasuwą Z9 odływu ze zbiorników do pompowni)
	//-----------------------------------------------------------------------------
	//Zmainy wprowadzone:
	//Wersja  Data       Osoba wprowadzająca zmiany - ekspert
	//01.00.00 11.05.2022 (Tecmer Radosław - twórca) Pieresza wersja 01.00.00
	//=============================================================================
	*)
	
	
	REGION otwieranie Z9
	  // jesli warunki spełnione
	  IF #isGotowość
	    AND #isAuto
	    AND #isREM
	    AND #isClose
	    AND ("DB10_instance_SCADA".TrybSterowania <> 0)
	    AND ("DB10_instance_SCADA".TrybSterowania <= 3)
	    
	  THEN
	    IF #isPumping OR #isRecharging OR #isAutPumping THEN
	      IF ("Hbit_Auto_Manu_Z1" AND "Hbit_Otwarta_Z1") OR ("Hbit_Auto_Manu_Z3" AND "Hbit_Otwarta_Z3") OR ( "Hbit_Auto_Manu_Z5" AND "Hbit_Otwarta_Z5") OR ("Hbit_Auto_Manu_Z7" AND"Hbit_Otwarta_Z7") THEN
	        // Otwieranie
	        #setSVMO := TRUE;
	      ELSE
	        #setSVMO := FALSE;
	        ;
	      END_IF;
	      
	      ;
	    END_IF;
	    
	    ;
	  END_IF;
	  
	END_REGION
	
	
	
	
	REGION zamykanie Z9 
	  // 
	  IF #isGotowość
	    AND #isAuto
	    AND #isClose = FALSE
	    AND #isREM
	    AND ("DB10_instance_SCADA".TrybSterowania <> 0)
	    AND ("DB10_instance_SCADA".TrybSterowania <= 3)
	    
	  THEN
	    IF "Zmienne_sterujące_zbiorników".Zbiornik_1.isEptying_Zb  = False
	      AND "Zmienne_sterujące_zbiorników".Zbiornik_2.isEptying_Zb = FALSE
	      AND "Zmienne_sterujące_zbiorników".Zbiornik_3.isEptying_Zb = FALSE
	      AND "Zmienne_sterujące_zbiorników".Zbiornik_4.isEptying_Zb = FALSE
	    THEN
	      // Zamykanie 
	      #setSVMC := TRUE;
	  ELSE
	    #setSVMC := FALSE;
	      ;
	    END_IF;
	    
	    
	    ;
	  END_IF;
	  
	  
	END_REGION
	
	
END_FUNCTION

FUNCTION "Sterowania _Zasuwa_Z10" : Void
TITLE = Sterowanie zasuwą Z9 odpływu ze zbiorników
{ S7_Optimized_Access := 'TRUE' }
AUTHOR : rtecmr
VERSION : 0.1
//Otwieranie zasuwy w cyklu przetłaczania, dosilania. PLC Pompownia na podstawie statusu zasuwy Z9 i bitu informującego o otwarciu rozoczyna procedurę przetłaczania lub dosilania
   VAR_INPUT 
      isGotowość : Bool;   // bit gotowości
      isAuto : Bool;   // bit trybu autoamt
      isOpen : Bool;   // potwierdzenia otwarta
      isClose : Bool;   // potwierdzenia zamknieta
      isFilling_zb1 : Bool;   // bit aktywacji napełniania zbiornika
      isFilling_zb2 : Bool;   // bit aktywacji napełniania zbiornika
      isFilling_zb3 : Bool;   // bit aktywacji napełniania zbiornika
      isFilling_zb4 : Bool;   // bit aktywacji napełniania zbiornika
      isREM : Bool;   // bit trybu automat
      "actValue-opening_Z10" : Int;   // Zmienna zapamietan w parametryzacji kontroli sterowaia zasuwą Z10
   END_VAR

   VAR_OUTPUT 
      setValue_opening_Z10 : Int;   // wartość zadana otwarcia Z10
      actOpen : Bool;   // bit aktywacji otwierania
      actClose : Bool;   // bit aktywacji zamykania
   END_VAR


BEGIN
	(*
	//=============================================================================
	//(JZWiK S.A Radosław Tecmer)
	//(c)Copyright (2022) All Rights Reserved
	//-----------------------------------------------------------------------------
	//Testowane z:   (system docelowy z  FW 4.4)
	//Pakiet inżynierski:   TIA Portal (V16 Update 5)
	//Ograniczenia:  ( - )
	//Wymagania:  (minimalne S7-1200 CPU 1215C FW 4.2 .)
	//Funkcjonalnośc: (Sterowanie zasuwą Z10 zasilającej zbiorniki. 
	                    Sterowanie sygnałem analogowym pozycji otwarci 0-100%)
	//-----------------------------------------------------------------------------
	//Zmainy wprowadzone:
	//Wersja  Data       Osoba wprowadzająca zmiany - ekspert
	//01.00.00 11.05.2022 (Tecmer Radosław - twórca) Pieresza wersja 01.00.00
	//=============================================================================
	*)
	
	
	REGION otwieranie Z10
	  // jesli warunki spełnione
	  IF #isGotowość
	    AND #isAuto
	    AND #isREM
	    AND #isClose
	    AND ("DB10_instance_SCADA".TrybSterowania <> 0)
	    AND ("DB10_instance_SCADA".TrybSterowania <= 3)
	    
	  THEN
	    IF #isFilling_zb1 OR #isFilling_zb2 OR #isFilling_zb3 OR #isFilling_zb4 THEN
	      IF "Hbit_Zamknieta_Z1" AND"Hbit_Zamknieta_Z3"AND"Hbit_Zamknieta_Z5"AND"Hbit_Zamknieta_Z7" THEN
	        // Otwieranie
	        #setValue_opening_Z10 := #"actValue-opening_Z10" ;
	        #actOpen := TRUE;
	      ELSE
	        #actOpen := FALSE;
	        ;
	      END_IF;
	      
	      ;
	    END_IF;
	    
	    ;
	  END_IF;
	  
	END_REGION
	
	
	
	
	REGION zamykanie Z10 
	  // 
	  IF #isGotowość
	    AND #isAuto
	    AND #isClose = FALSE
	    AND #isREM
	    AND ("DB10_instance_SCADA".TrybSterowania <> 0)
	    AND ("DB10_instance_SCADA".TrybSterowania <= 3)
	    
	  THEN
	    IF #isFilling_zb1  = False
	      AND #isFilling_zb2 = FALSE
	      AND #isFilling_zb3 = FALSE
	      AND #isFilling_zb4 = FALSE
	    THEN
	      // Zamykanie 
	      #setValue_opening_Z10 := 0 ;
	      #actClose := TRUE;
	  ELSE
	    #actClose := FALSE;
	    
	      ;
	    END_IF;
	    
	    
	    ;
	  END_IF;
	  
	  
	END_REGION
	
	
END_FUNCTION

FUNCTION_BLOCK "Byte Status Z1-Z10"
TITLE = Status napędów
{ S7_Optimized_Access := 'TRUE' }
AUTHOR : rtecmer
VERSION : 0.1
//Funkcja kompije status napędu z instancji DB10 do znaczników.
//Persowanie danych napędów.

BEGIN
	(*
	//=============================================================================
	//(JZWiK S.A Radosław Tecmer)
	//(c)Copyright (2021) All Rights Reserved
	//-----------------------------------------------------------------------------
	//Testowane z:   (system docelowy z  FW 4.4)
	//Pakiet inżynierski:   TIA Portal (V14 Sp1 Update 9)
	//Ograniczenia:  ( - )
	//Wymagania:  (minimalne S7-1200 CPU 1215C FW 4.2 .)
	//Funkcjonalnośc: (Byte statusu napędów Zasuw Z1-Z10 )
	//-----------------------------------------------------------------------------
	//Zmainy wprowadzone:
	//Wersja  Data       Osoba wprowadzająca zmiany - ekspert
	//01.00.00 17.11.2021 (Tecmer Radosław - twórca) Pieresza wersja 01.00.00
	//=============================================================================
	*)
	
	REGION Status Zasuw
	  // przekazanie wartości wartości z DB10 do słowa znacznika
	  "Byte_Status_Z1" := "DB10_instance_SCADA".instZ1;
	  "Byte_Status_Z2" := "DB10_instance_SCADA".instZ2;
	  "Byte_Status_Z3" := "DB10_instance_SCADA".instZ3;
	  "Byte_Status_Z4" := "DB10_instance_SCADA".instZ4;
	  "Byte_Status_Z5" := "DB10_instance_SCADA".instZ5;
	  "Byte_Status_Z6" := "DB10_instance_SCADA".instZ6;
	  "Byte_Status_Z7" := "DB10_instance_SCADA".instZ7;
	  "Byte_Status_Z8" := "DB10_instance_SCADA".instZ8;
	  "Byte_Status_Z9" := "DB10_instance_SCADA".instZ9;
	  "Byte_Status_Z10" := "DB10_instance_SCADA".instZ10;
	  
	  
	END_REGION
	
END_FUNCTION_BLOCK

FUNCTION "Alarmy" : Void
TITLE = KOntrola zabezpieczen momentowych
{ S7_Optimized_Access := 'TRUE' }
AUTHOR : rtecmer
VERSION : 0.1
//Jesli obwód przerwany to błąd od momentu

BEGIN
	(*
	//=============================================================================
	//(JZWiK S.A Radosław Tecmer)
	//(c)Copyright (2022) All Rights Reserved
	//-----------------------------------------------------------------------------
	//Testowane z:   (system docelowy z  FW 4.4)
	//Pakiet inżynierski:   TIA Portal (V16 Update 5)
	//Ograniczenia:  ( - )
	//Wymagania:  (minimalne S7-1200 CPU 1215C FW 4.2 .)
	//Funkcjonalnośc: (Kontrola awarii od sytku momoentowego napędu )
	//-----------------------------------------------------------------------------
	//Zmainy wprowadzone:
	//Wersja  Data       Osoba wprowadzająca zmiany - ekspert
	//01.00.00 09.03.2022 (Tecmer Radosław - twórca) Pieresza wersja 01.00.00
	//=============================================================================
	*)
	
	REGION przekazanie do db stan styków momentowych Z1 - Z9
	  // przekazywanie stanu stykuów dla wszystkich napedów
	  %DB10.DBX69.0 := "setAlarm_Moment_Z_1";
	  %DB10.DBX69.1 := "setAlarm_Moment_Z_2";
	  %DB10.DBX69.2 := "setAlarm_Moment_Z_3";
	  %DB10.DBX69.3 := "setAlarm_Moment_Z_4";
	  %DB10.DBX69.4 := "setAlarm_Moment_Z_5";
	  %DB10.DBX69.5 := "setAlarm_Moment_Z_6";
	  %DB10.DBX69.6 := "setAlarm_Moment_Z_7";
	  %DB10.DBX69.7 := "setAlarm_Moment_Z_8";
	  %DB10.DBX68.7 := "setAlarm_Moment_Z_9";
	  %DB10.DBX68.6 := "setAlarm_Moment_Z_10";
	  
	  
	END_REGION
	
	
	REGION Z1
	  // styk momentu
	  IF "inputAwariaMomentZ_1" = False THEN
	    // ustaw alarm
	    "setAlarm_Moment_Z_1" := TRUE;
	  ELSE
	    "setAlarm_Moment_Z_1" := FALSE;
	    ;
	  END_IF;
	  
	END_REGION
	
	REGION Z2
	  // styk momentu
	  IF "inputAwariaMomentZ_2" = False THEN
	    // ustaw alarm
	    "setAlarm_Moment_Z_2" := TRUE;
	  ELSE
	    "setAlarm_Moment_Z_2" := FALSE
	    ;
	  END_IF;
	  
	END_REGION
	
	REGION Z3
	  // styk momentu
	  IF "inputAwariaMomentZ_3" = False THEN
	    // ustaw alarm
	    "setAlarm_Moment_Z_3" := TRUE;
	  ELSE
	    "setAlarm_Moment_Z_3" := FALSE
	    ;
	  END_IF;
	  
	END_REGION
	
	REGION Z4
	  // styk momentu
	  IF "inputAwariaMomentZ_4" = False THEN
	    // ustaw alarm
	    "setAlarm_Moment_Z_4" := TRUE;
	  ELSE
	    "setAlarm_Moment_Z_4" := FALSE
	    ;
	  END_IF;
	  
	END_REGION
	
	REGION Z5
	  // styk momentu
	  IF "inputAwariaMomentZ_5" = False THEN
	    // ustaw alarm
	    "setAlarm_Moment_Z_5" := TRUE;
	  ELSE
	    "setAlarm_Moment_Z_5" := FALSE
	    ;
	  END_IF;
	  
	END_REGION
	
	REGION Z6
	  // styk momentu
	  IF "inputAwariaMomentZ_6" = False THEN
	    // ustaw alarm
	    "setAlarm_Moment_Z_6" := TRUE;
	  ELSE
	    "setAlarm_Moment_Z_6" := FALSE
	    ;
	  END_IF;
	  
	END_REGION
	
	REGION Z7
	  // styk momentu
	  IF "inputAwariaMomentZ_7" = False THEN
	    // ustaw alarm
	    "setAlarm_Moment_Z_7" := TRUE;
	  ELSE
	    "setAlarm_Moment_Z_7" := FALSE
	    ;
	  END_IF;
	  
	END_REGION
	
	REGION Z8
	  // styk momentu
	  IF "inputAwariaMomentZ_8" = False THEN
	    // ustaw alarm
	    "setAlarm_Moment_Z_8" := TRUE;
	  ELSE
	    "setAlarm_Moment_Z_8" := FALSE
	    ;
	  END_IF;
	  
	END_REGION
	
	REGION Z9
	  // styk momentu
	  IF "inputAwariaMomentZ_9" = False THEN
	    // ustaw alarm
	    "setAlarm_Moment_Z_9" := TRUE;
	  ELSE
	    "setAlarm_Moment_Z_9" := FALSE
	    ;
	  END_IF;
	  
	END_REGION
	
	
	
	REGION Alarm zbiorczy napedów 
	  //Z1
	  IF "isGotowość_Z_1" =  FALSE THEN
	    // ustaw sygnał awarii
	    %DB10.DBX6.0 := TRUE;
	    %DB10.DBX7.0 := TRUE;
	    
	
	    ;
	  END_IF;
	  
	  //Z2
	  IF "isGotowość_Z_2" = FALSE THEN
	    // ustaw sygnał awarii
	    %DB10.DBX8.0 := TRUE;
	    %DB10.DBX9.0 := TRUE;
	    
	    ;
	  END_IF;
	  
	
	  //Z3
	  IF "isGotowość_Z_3" = FALSE THEN
	    // ustaw sygnał awarii
	    %DB10.DBX10.0 := TRUE;
	    %DB10.DBX11.0 := TRUE;
	   
	    ;
	  END_IF;
	  
	  //Z4
	  IF "isGotowość_Z_4" = FALSE THEN
	    // ustaw sygnał awarii
	    %DB10.DBX12.0 := TRUE;
	    %DB10.DBX13.0 := TRUE;
	   
	    ;
	  END_IF;
	  
	
	  //Z5
	  IF "isGotowość_Z_5" = FALSE THEN
	    // ustaw sygnał awarii
	    %DB10.DBX14.0 := TRUE;
	    %DB10.DBX15.0 := TRUE;
	    
	    ;
	  END_IF;
	  
	  //Z6
	  IF "isGotowość_Z_6" = FALSE THEN
	    // ustaw sygnał awarii
	    %DB10.DBX16.0 := TRUE;
	    %DB10.DBX17.0 := TRUE;
	   
	    ;
	  END_IF;
	  
	  //Z7
	  IF "isGotowość_Z_7" = FALSE THEN
	    // ustaw sygnał awarii
	    %DB10.DBX18.0 := TRUE;
	    %DB10.DBX19.0 := TRUE;
	    
	    ;
	  END_IF;
	  
	  //Z8
	  IF "isGotowość_Z_8" = FALSE THEN
	    // ustaw sygnał awarii
	    %DB10.DBX20.0 := TRUE;
	    %DB10.DBX21.0 := TRUE;
	   
	    ;
	  END_IF;
	  
	
	  //Z9
	  IF "isGotowość_Z_9" = FALSE THEN
	    // ustaw sygnał awarii
	    %DB10.DBX22.0 := TRUE;
	    %DB10.DBX23.0 := TRUE;
	    
	    
	    ;
	  END_IF;
	  
	  //Z10
	  IF "isGotowość_Z_10" =  FALSE THEN
	    // ustaw sygnał awarii
	    %DB10.DBX24.0 := TRUE;
	    %DB10.DBX25.0 := TRUE;
	    
	    
	    ;
	  END_IF;
	  
	
	  
	  
	END_REGION
	
	REGION Modbus RTU Q1 przepływomierz Zasuwy
	  // Jeśli błąd komunikacji to zerowanie przepływu chwilowego
	  
	  IF "dbTags_master_MPP04_2".modbusMaster.errorStatus <> 0 THEN
	    // zerwowanie przepływu
	    "dbMasterData".data6_Wielkość_przeływu_Adres_0.data[0] := 0;
	    "dbMasterData".data6_Wielkość_przeływu_Adres_0.data[1] := 0
	    ;
	  END_IF;
	  
	END_REGION
	
	REGION HMI info alarmy
	  // gdy w cyklu napełniania wystąpi alarm od niskiego ciśnienia na magistrali
	  IF "setAlarmNiskie_magistrala" AND ("HMI.Filing1"
	    OR "HMI.Filing2"  //jest czas na napełnianie
	    OR "HMI.Filing3"  //jest czas na napełnianie
	    OR "HMI.Filing4") //jest czas na napełnianie
	  THEN
	    // ustaw bit informacji do HMI przerwane napełnianie 
	    "HMI.StopFiling" := True;
	  ELSE
	    "HMI.StopFiling" := FALSE
	    ;
	  END_IF;
	  
	  
	END_REGION
	
	
	
	
	
	
	
	
	
	
END_FUNCTION

FUNCTION "Zmienne_SCADA" : Void
{ S7_Optimized_Access := 'TRUE' }
VERSION : 0.1

BEGIN
	(*
	//=============================================================================
	//(JZWiK S.A Radosław Tecmer)
	//(c)Copyright (2021) All Rights Reserved
	//-----------------------------------------------------------------------------
	//Testowane z:   (system docelowy z  FW 4.2)
	//Pakiet inżynierski:   TIA Portal (V14 Sp1 Update 9)
	//Ograniczenia:  ( - )
	//Wymagania:  (minimalne S7-1200 CPU 1214 FW 3.2 .)
	//Funkcjonalnośc: (Kopiowanie bloków danych z - do bloku SCADA )
	//-----------------------------------------------------------------------------
	//Zmainy wprowadzone:
	//Wersja  Data       Osoba wprowadzająca zmiany - ekspert
	//01.00.00 28.01.2022 (Tecmer Radosław - twórca) Pieresza wersja 01.00.00
	//=============================================================================
	*)
	
	//
	
	
	
	REGION Przepływomierz
	  
	  IF "switch_flow_analog_modbus" THEN
	    // jeśli True to analog
	    "DB10_instance_SCADA".actPrzepływ_Q2 := "dbdane".Wielkość_przepływu_Q2_analog;
	    
	  ELSE
	    // jeśli  False to modbus rtu
	    "DB10_instance_SCADA".actPrzepływ_Q2 := "dbdane".Wielkość_przeływu_Q2;
	    ;
	  END_IF;
	  
	  // 
	  "DB10_instance_SCADA".sumPrzepływVF_Q2 := "dbdane".Licznik_objętość_VF_Q2;
	  "DB10_instance_SCADA".statusPrzepływVR_Q2 := "dbdane"._Stan_urządzenia_Q2;
	END_REGION
	
	REGION Z10 - położenie
	  // aktualna wartość
	  "DB10_instance_SCADA".actPołożenieZ10 :="dbtags_Sterowanie"."Z10 Pozycja".encoder;
	  
	END_REGION
	
	
	
	
	REGION Modbus RTU przekazanie kodu błędu 
	  // Statement section REGION
	  "DB10_instance_SCADA".rtu_mpp04_2error_status := "dbTags_master_MPP04_2".modbusMaster.errorStatus;
	END_REGION
	
	// Pompownia
	REGION Strategia sterowania pompownią
	  // strategia
	  "DB10_instance_SCADA".ModelSterowania := "dbHold_download".sterowanie.set_strategia_sterowania;
	  
	END_REGION
	
	
	(*
	Przekazanie wartości analogowych CIŚNIENIE, ZBIORNIKI  z wyborem z filtracją Kolmana / bez
	*)
	REGION Analogi ciśnienie B5 i poziom w zbiornikach
	  // 
	  IF "switch_Kolman" THEN
	    // przekaż wartość bezpośrednie z analogów 
	    "DB10_instance_SCADA"."actCiśnienie-magistralaB5" := "dbtags_Sterowanie"."Analog pomiar".AI_ciśnienie_B5;
	    "DB10_instance_SCADA".actPoziomZbiornik_1 := "dbtags_Sterowanie"."Analog pomiar".AI_poziom_zbiornik_1;
	    "DB10_instance_SCADA".actPoziomZbiornik_2 := "dbtags_Sterowanie"."Analog pomiar".AI_poziom_zbiornik_2;
	    "DB10_instance_SCADA".actPoziomZbiornik_3 := "dbtags_Sterowanie"."Analog pomiar".AI_poziom_zbiornik_3;
	    "DB10_instance_SCADA".actPoziomZbiornik_4 := "dbtags_Sterowanie"."Analog pomiar".AI_poziom_zbiornik_4;
	   
	  ELSE
	    //przekaż wartość po filtracji Kolmana
	    "DB10_instance_SCADA"."actCiśnienie-magistralaB5" := "dbtags_Sterowanie"."Analog pomiar".AI_ciśnienie_B5;
	    "DB10_instance_SCADA".actPoziomZbiornik_1 := "dbtags_Sterowanie"."Analog pomiar".kolman_poziom_zbiornik_1;
	    "DB10_instance_SCADA".actPoziomZbiornik_2 := "dbtags_Sterowanie"."Analog pomiar".kolman_poziom_zbiornik_2;
	    "DB10_instance_SCADA".actPoziomZbiornik_3 := "dbtags_Sterowanie"."Analog pomiar".kolman_poziom_zbiornik_3;
	    "DB10_instance_SCADA".actPoziomZbiornik_4 := "dbtags_Sterowanie"."Analog pomiar".kolman_poziom_zbiornik_4;
	    
	    ;
	  END_IF;
	  
	  
	END_REGION
	
	// wartość alarmowa ciśnienia magistrala B5 ustawiana z PLC pompownia
	"Parametryzacja"."Setting Controll".alarmMin_CiśnienieGranica := "dbHold_download".sterowanie.set_magistrala_alarm_min_bar;
	
	  
	  
	
	
	
	
END_FUNCTION

FUNCTION "Synchroniczna_wymiana_danych_PLC1-PLC2" : Void   // FC34, LAD
TITLE = Przekazywanie zmian parametrów
{ S7_Optimized_Access := 'TRUE' }
AUTHOR : rtecmer
VERSION : 0.1
// Funkcja grupuje bloki funkcji służąc wymianie danych HMI - PLC1, HMI-PLC2 i SCADA. Wprowadzanie wartości z poziomu HMI Zbiorniki lub HMI Pompownia czy SCADA jest nadpisywane w docelowym sterowniku. Zmian włónych parametrów układu sterowania pompownią, zbiornikami można dokonywać w dowolnego miejsca.
// stored: AutoNumber true, IsIECCheckEnabled false, SetENOAutomatically false, UDAEnableTagReadback false
   VAR_TEMP   // added for the SCL form of the ladder/FBD networks
      _w1 : Bool;
   END_VAR
BEGIN

REGION Network 2: Detekcja zmiany wartości nastaw - Pozim napełniania
   // Funkcja po przeprowadzeniu sprawdzenia czy nastąpiły zmiany w danych przekazuje nowe wartości
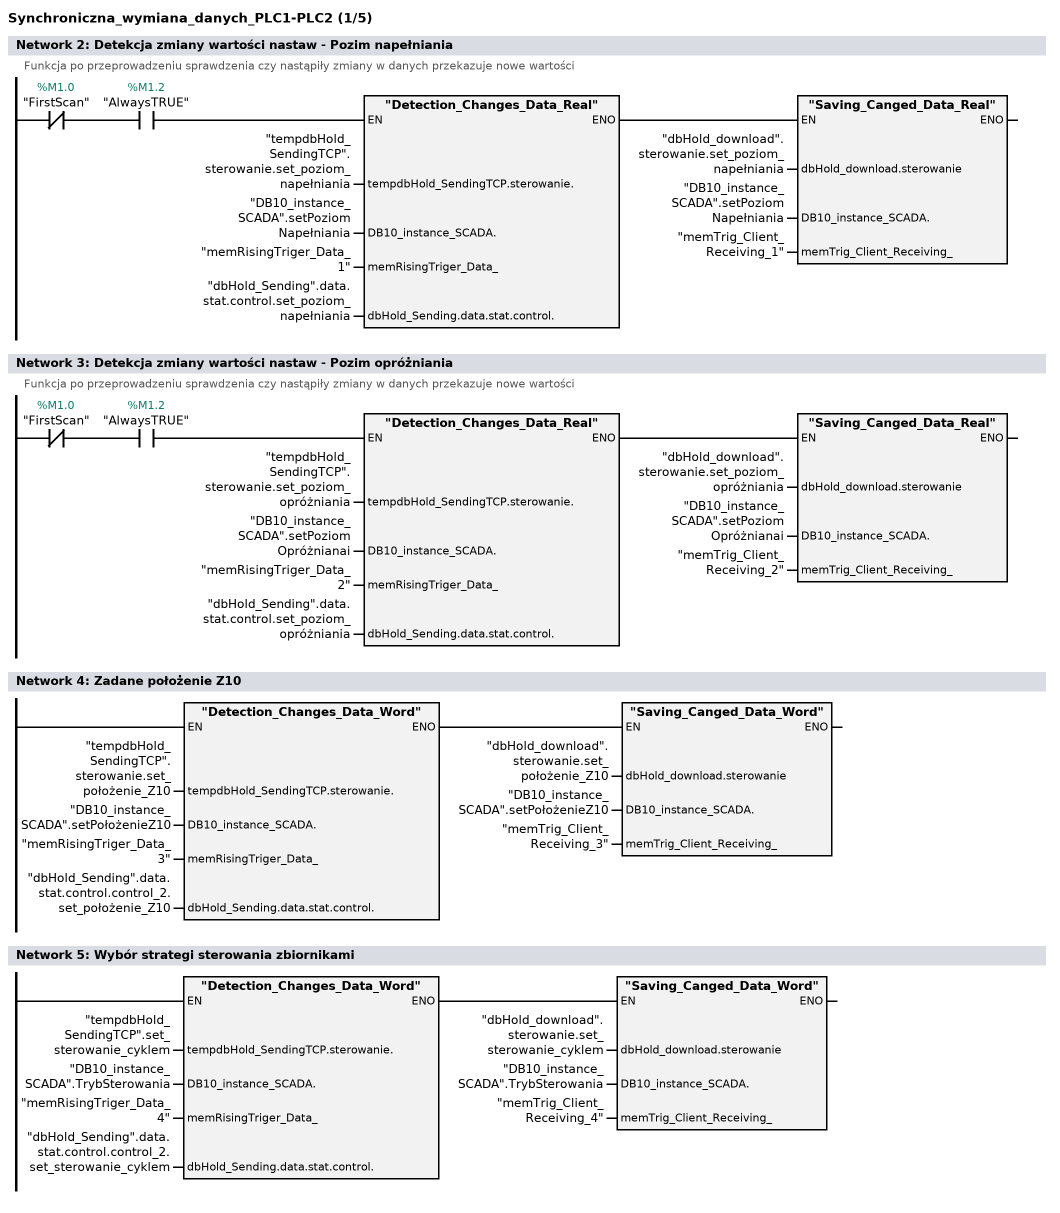
   RUNG wire#powerrail
      I_Contact( "FirstScan" )
      Contact( "AlwaysTRUE" )
      "Detection_Changes_Data_Real"("tempdbHold_SendingTCP.sterowanie." := "tempdbHold_SendingTCP".sterowanie.set_poziom_napełniania, "DB10_instance_SCADA." := "DB10_instance_SCADA".setPoziomNapełniania, memRisingTriger_Data_ := "memRisingTriger_Data_1", "dbHold_Sending.data.stat.control." := "dbHold_Sending".data.stat.control.set_poziom_napełniania)
      "Saving_Canged_Data_Real"("dbHold_download.sterowanie" := "dbHold_download".sterowanie.set_poziom_napełniania, "DB10_instance_SCADA." := "DB10_instance_SCADA".setPoziomNapełniania, memTrig_Client_Receiving_ := "memTrig_Client_Receiving_1")
   END_RUNG
   // the same network as SCL:
   "Detection_Changes_Data_Real"(EN := NOT "FirstScan" AND "AlwaysTRUE",
                           "tempdbHold_SendingTCP.sterowanie." := "tempdbHold_SendingTCP".sterowanie.set_poziom_napełniania,
                           "DB10_instance_SCADA." := "DB10_instance_SCADA".setPoziomNapełniania,
                           memRisingTriger_Data_ := "memRisingTriger_Data_1",
                           "dbHold_Sending.data.stat.control." := "dbHold_Sending".data.stat.control.set_poziom_napełniania,
                           ENO => #_w1);
   IF #_w1 THEN
       "Saving_Canged_Data_Real"("dbHold_download.sterowanie" := "dbHold_download".sterowanie.set_poziom_napełniania,
                               "DB10_instance_SCADA." := "DB10_instance_SCADA".setPoziomNapełniania,
                               memTrig_Client_Receiving_ := "memTrig_Client_Receiving_1");
   END_IF;
END_REGION

REGION Network 3: Detekcja zmiany wartości nastaw - Pozim opróżniania
   // Funkcja po przeprowadzeniu sprawdzenia czy nastąpiły zmiany w danych przekazuje nowe wartości
   RUNG wire#powerrail
      I_Contact( "FirstScan" )
      Contact( "AlwaysTRUE" )
      "Detection_Changes_Data_Real"("tempdbHold_SendingTCP.sterowanie." := "tempdbHold_SendingTCP".sterowanie.set_poziom_opróżniania, "DB10_instance_SCADA." := "DB10_instance_SCADA".setPoziomOpróżnianai, memRisingTriger_Data_ := "memRisingTriger_Data_2", "dbHold_Sending.data.stat.control." := "dbHold_Sending".data.stat.control.set_poziom_opróżniania)
      "Saving_Canged_Data_Real"("dbHold_download.sterowanie" := "dbHold_download".sterowanie.set_poziom_opróżniania, "DB10_instance_SCADA." := "DB10_instance_SCADA".setPoziomOpróżnianai, memTrig_Client_Receiving_ := "memTrig_Client_Receiving_2")
   END_RUNG
   // the same network as SCL:
   "Detection_Changes_Data_Real"(EN := NOT "FirstScan" AND "AlwaysTRUE",
                           "tempdbHold_SendingTCP.sterowanie." := "tempdbHold_SendingTCP".sterowanie.set_poziom_opróżniania,
                           "DB10_instance_SCADA." := "DB10_instance_SCADA".setPoziomOpróżnianai,
                           memRisingTriger_Data_ := "memRisingTriger_Data_2",
                           "dbHold_Sending.data.stat.control." := "dbHold_Sending".data.stat.control.set_poziom_opróżniania,
                           ENO => #_w1);
   IF #_w1 THEN
       "Saving_Canged_Data_Real"("dbHold_download.sterowanie" := "dbHold_download".sterowanie.set_poziom_opróżniania,
                               "DB10_instance_SCADA." := "DB10_instance_SCADA".setPoziomOpróżnianai,
                               memTrig_Client_Receiving_ := "memTrig_Client_Receiving_2");
   END_IF;
END_REGION

REGION Network 4: Zadane położenie Z10
   RUNG wire#powerrail
      "Detection_Changes_Data_Word"("tempdbHold_SendingTCP.sterowanie." := "tempdbHold_SendingTCP".sterowanie.set_położenie_Z10, "DB10_instance_SCADA." := "DB10_instance_SCADA".setPołożenieZ10, memRisingTriger_Data_ := "memRisingTriger_Data_3", "dbHold_Sending.data.stat.control." := "dbHold_Sending".data.stat.control.control_2.set_położenie_Z10)
      "Saving_Canged_Data_Word"("dbHold_download.sterowanie" := "dbHold_download".sterowanie.set_położenie_Z10, "DB10_instance_SCADA." := "DB10_instance_SCADA".setPołożenieZ10, memTrig_Client_Receiving_ := "memTrig_Client_Receiving_3")
   END_RUNG
   // the same network as SCL:
   "Detection_Changes_Data_Word"("tempdbHold_SendingTCP.sterowanie." := "tempdbHold_SendingTCP".sterowanie.set_położenie_Z10,
                           "DB10_instance_SCADA." := "DB10_instance_SCADA".setPołożenieZ10,
                           memRisingTriger_Data_ := "memRisingTriger_Data_3",
                           "dbHold_Sending.data.stat.control." := "dbHold_Sending".data.stat.control.control_2.set_położenie_Z10,
                           ENO => #_w1);
   IF #_w1 THEN
       "Saving_Canged_Data_Word"("dbHold_download.sterowanie" := "dbHold_download".sterowanie.set_położenie_Z10,
                               "DB10_instance_SCADA." := "DB10_instance_SCADA".setPołożenieZ10,
                               memTrig_Client_Receiving_ := "memTrig_Client_Receiving_3");
   END_IF;
END_REGION

REGION Network 5: Wybór strategi sterowania zbiornikami
   RUNG wire#powerrail
      "Detection_Changes_Data_Word"("tempdbHold_SendingTCP.sterowanie." := "tempdbHold_SendingTCP".set_sterowanie_cyklem, "DB10_instance_SCADA." := "DB10_instance_SCADA".TrybSterowania, memRisingTriger_Data_ := "memRisingTriger_Data_4", "dbHold_Sending.data.stat.control." := "dbHold_Sending".data.stat.control.control_2.set_sterowanie_cyklem)
      "Saving_Canged_Data_Word"("dbHold_download.sterowanie" := "dbHold_download".sterowanie.set_sterowanie_cyklem, "DB10_instance_SCADA." := "DB10_instance_SCADA".TrybSterowania, memTrig_Client_Receiving_ := "memTrig_Client_Receiving_4")
   END_RUNG
   // the same network as SCL:
   "Detection_Changes_Data_Word"("tempdbHold_SendingTCP.sterowanie." := "tempdbHold_SendingTCP".set_sterowanie_cyklem,
                           "DB10_instance_SCADA." := "DB10_instance_SCADA".TrybSterowania,
                           memRisingTriger_Data_ := "memRisingTriger_Data_4",
                           "dbHold_Sending.data.stat.control." := "dbHold_Sending".data.stat.control.control_2.set_sterowanie_cyklem,
                           ENO => #_w1);
   IF #_w1 THEN
       "Saving_Canged_Data_Word"("dbHold_download.sterowanie" := "dbHold_download".sterowanie.set_sterowanie_cyklem,
                               "DB10_instance_SCADA." := "DB10_instance_SCADA".TrybSterowania,
                               memTrig_Client_Receiving_ := "memTrig_Client_Receiving_4");
   END_IF;
END_REGION

REGION Network 6: Godzina start napełnianie
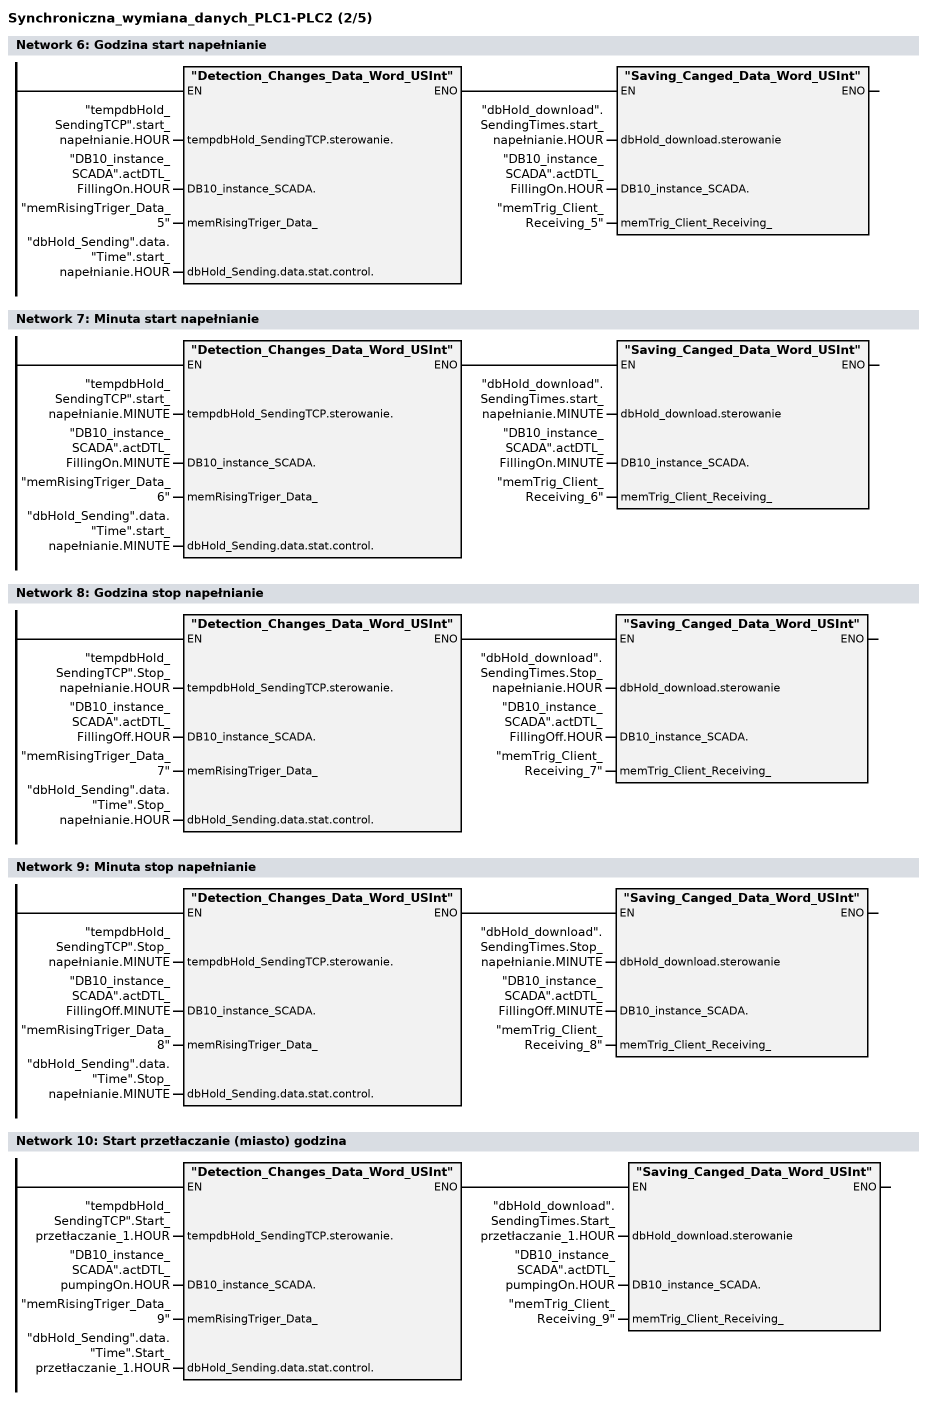
   RUNG wire#powerrail
      "Detection_Changes_Data_Word_USInt"("tempdbHold_SendingTCP.sterowanie." := "tempdbHold_SendingTCP".start_napełnianie.HOUR, "DB10_instance_SCADA." := "DB10_instance_SCADA".actDTL_FillingOn.HOUR, memRisingTriger_Data_ := "memRisingTriger_Data_5", "dbHold_Sending.data.stat.control." := "dbHold_Sending".data."Time".start_napełnianie.HOUR)
      "Saving_Canged_Data_Word_USInt"("dbHold_download.sterowanie" := "dbHold_download".SendingTimes.start_napełnianie.HOUR, "DB10_instance_SCADA." := "DB10_instance_SCADA".actDTL_FillingOn.HOUR, memTrig_Client_Receiving_ := "memTrig_Client_Receiving_5")
   END_RUNG
   // the same network as SCL:
   "Detection_Changes_Data_Word_USInt"("tempdbHold_SendingTCP.sterowanie." := "tempdbHold_SendingTCP".start_napełnianie.HOUR,
                           "DB10_instance_SCADA." := "DB10_instance_SCADA".actDTL_FillingOn.HOUR,
                           memRisingTriger_Data_ := "memRisingTriger_Data_5",
                           "dbHold_Sending.data.stat.control." := "dbHold_Sending".data."Time".start_napełnianie.HOUR,
                           ENO => #_w1);
   IF #_w1 THEN
       "Saving_Canged_Data_Word_USInt"("dbHold_download.sterowanie" := "dbHold_download".SendingTimes.start_napełnianie.HOUR,
                               "DB10_instance_SCADA." := "DB10_instance_SCADA".actDTL_FillingOn.HOUR,
                               memTrig_Client_Receiving_ := "memTrig_Client_Receiving_5");
   END_IF;
END_REGION

REGION Network 7: Minuta start napełnianie
   RUNG wire#powerrail
      "Detection_Changes_Data_Word_USInt"("tempdbHold_SendingTCP.sterowanie." := "tempdbHold_SendingTCP".start_napełnianie.MINUTE, "DB10_instance_SCADA." := "DB10_instance_SCADA".actDTL_FillingOn.MINUTE, memRisingTriger_Data_ := "memRisingTriger_Data_6", "dbHold_Sending.data.stat.control." := "dbHold_Sending".data."Time".start_napełnianie.MINUTE)
      "Saving_Canged_Data_Word_USInt"("dbHold_download.sterowanie" := "dbHold_download".SendingTimes.start_napełnianie.MINUTE, "DB10_instance_SCADA." := "DB10_instance_SCADA".actDTL_FillingOn.MINUTE, memTrig_Client_Receiving_ := "memTrig_Client_Receiving_6")
   END_RUNG
   // the same network as SCL:
   "Detection_Changes_Data_Word_USInt"("tempdbHold_SendingTCP.sterowanie." := "tempdbHold_SendingTCP".start_napełnianie.MINUTE,
                           "DB10_instance_SCADA." := "DB10_instance_SCADA".actDTL_FillingOn.MINUTE,
                           memRisingTriger_Data_ := "memRisingTriger_Data_6",
                           "dbHold_Sending.data.stat.control." := "dbHold_Sending".data."Time".start_napełnianie.MINUTE,
                           ENO => #_w1);
   IF #_w1 THEN
       "Saving_Canged_Data_Word_USInt"("dbHold_download.sterowanie" := "dbHold_download".SendingTimes.start_napełnianie.MINUTE,
                               "DB10_instance_SCADA." := "DB10_instance_SCADA".actDTL_FillingOn.MINUTE,
                               memTrig_Client_Receiving_ := "memTrig_Client_Receiving_6");
   END_IF;
END_REGION

REGION Network 8: Godzina stop napełnianie
   RUNG wire#powerrail
      "Detection_Changes_Data_Word_USInt"("tempdbHold_SendingTCP.sterowanie." := "tempdbHold_SendingTCP".Stop_napełnianie.HOUR, "DB10_instance_SCADA." := "DB10_instance_SCADA".actDTL_FillingOff.HOUR, memRisingTriger_Data_ := "memRisingTriger_Data_7", "dbHold_Sending.data.stat.control." := "dbHold_Sending".data."Time".Stop_napełnianie.HOUR)
      "Saving_Canged_Data_Word_USInt"("dbHold_download.sterowanie" := "dbHold_download".SendingTimes.Stop_napełnianie.HOUR, "DB10_instance_SCADA." := "DB10_instance_SCADA".actDTL_FillingOff.HOUR, memTrig_Client_Receiving_ := "memTrig_Client_Receiving_7")
   END_RUNG
   // the same network as SCL:
   "Detection_Changes_Data_Word_USInt"("tempdbHold_SendingTCP.sterowanie." := "tempdbHold_SendingTCP".Stop_napełnianie.HOUR,
                           "DB10_instance_SCADA." := "DB10_instance_SCADA".actDTL_FillingOff.HOUR,
                           memRisingTriger_Data_ := "memRisingTriger_Data_7",
                           "dbHold_Sending.data.stat.control." := "dbHold_Sending".data."Time".Stop_napełnianie.HOUR,
                           ENO => #_w1);
   IF #_w1 THEN
       "Saving_Canged_Data_Word_USInt"("dbHold_download.sterowanie" := "dbHold_download".SendingTimes.Stop_napełnianie.HOUR,
                               "DB10_instance_SCADA." := "DB10_instance_SCADA".actDTL_FillingOff.HOUR,
                               memTrig_Client_Receiving_ := "memTrig_Client_Receiving_7");
   END_IF;
END_REGION

REGION Network 9: Minuta stop napełnianie
   RUNG wire#powerrail
      "Detection_Changes_Data_Word_USInt"("tempdbHold_SendingTCP.sterowanie." := "tempdbHold_SendingTCP".Stop_napełnianie.MINUTE, "DB10_instance_SCADA." := "DB10_instance_SCADA".actDTL_FillingOff.MINUTE, memRisingTriger_Data_ := "memRisingTriger_Data_8", "dbHold_Sending.data.stat.control." := "dbHold_Sending".data."Time".Stop_napełnianie.MINUTE)
      "Saving_Canged_Data_Word_USInt"("dbHold_download.sterowanie" := "dbHold_download".SendingTimes.Stop_napełnianie.MINUTE, "DB10_instance_SCADA." := "DB10_instance_SCADA".actDTL_FillingOff.MINUTE, memTrig_Client_Receiving_ := "memTrig_Client_Receiving_8")
   END_RUNG
   // the same network as SCL:
   "Detection_Changes_Data_Word_USInt"("tempdbHold_SendingTCP.sterowanie." := "tempdbHold_SendingTCP".Stop_napełnianie.MINUTE,
                           "DB10_instance_SCADA." := "DB10_instance_SCADA".actDTL_FillingOff.MINUTE,
                           memRisingTriger_Data_ := "memRisingTriger_Data_8",
                           "dbHold_Sending.data.stat.control." := "dbHold_Sending".data."Time".Stop_napełnianie.MINUTE,
                           ENO => #_w1);
   IF #_w1 THEN
       "Saving_Canged_Data_Word_USInt"("dbHold_download.sterowanie" := "dbHold_download".SendingTimes.Stop_napełnianie.MINUTE,
                               "DB10_instance_SCADA." := "DB10_instance_SCADA".actDTL_FillingOff.MINUTE,
                               memTrig_Client_Receiving_ := "memTrig_Client_Receiving_8");
   END_IF;
END_REGION

REGION Network 10: Start przetłaczanie (miasto) godzina
   RUNG wire#powerrail
      "Detection_Changes_Data_Word_USInt"("tempdbHold_SendingTCP.sterowanie." := "tempdbHold_SendingTCP".Start_przetłaczanie_1.HOUR, "DB10_instance_SCADA." := "DB10_instance_SCADA".actDTL_pumpingOn.HOUR, memRisingTriger_Data_ := "memRisingTriger_Data_9", "dbHold_Sending.data.stat.control." := "dbHold_Sending".data."Time".Start_przetłaczanie_1.HOUR)
      "Saving_Canged_Data_Word_USInt"("dbHold_download.sterowanie" := "dbHold_download".SendingTimes.Start_przetłaczanie_1.HOUR, "DB10_instance_SCADA." := "DB10_instance_SCADA".actDTL_pumpingOn.HOUR, memTrig_Client_Receiving_ := "memTrig_Client_Receiving_9")
   END_RUNG
   // the same network as SCL:
   "Detection_Changes_Data_Word_USInt"("tempdbHold_SendingTCP.sterowanie." := "tempdbHold_SendingTCP".Start_przetłaczanie_1.HOUR,
                           "DB10_instance_SCADA." := "DB10_instance_SCADA".actDTL_pumpingOn.HOUR,
                           memRisingTriger_Data_ := "memRisingTriger_Data_9",
                           "dbHold_Sending.data.stat.control." := "dbHold_Sending".data."Time".Start_przetłaczanie_1.HOUR,
                           ENO => #_w1);
   IF #_w1 THEN
       "Saving_Canged_Data_Word_USInt"("dbHold_download.sterowanie" := "dbHold_download".SendingTimes.Start_przetłaczanie_1.HOUR,
                               "DB10_instance_SCADA." := "DB10_instance_SCADA".actDTL_pumpingOn.HOUR,
                               memTrig_Client_Receiving_ := "memTrig_Client_Receiving_9");
   END_IF;
END_REGION

REGION Network 11: Start przetłaczanie (miasto) mnutya
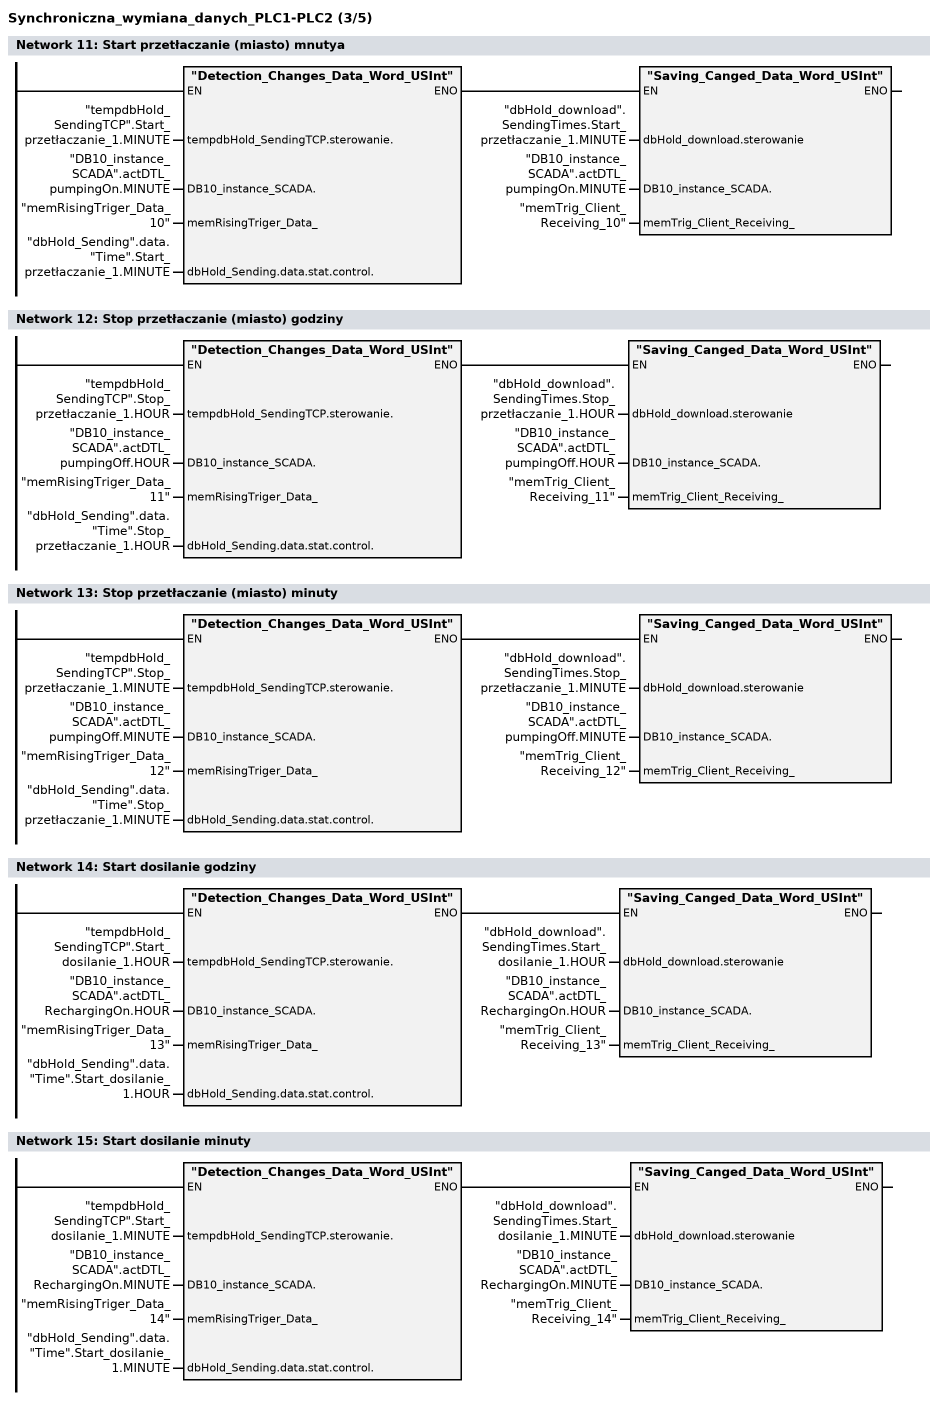
   RUNG wire#powerrail
      "Detection_Changes_Data_Word_USInt"("tempdbHold_SendingTCP.sterowanie." := "tempdbHold_SendingTCP".Start_przetłaczanie_1.MINUTE, "DB10_instance_SCADA." := "DB10_instance_SCADA".actDTL_pumpingOn.MINUTE, memRisingTriger_Data_ := "memRisingTriger_Data_10", "dbHold_Sending.data.stat.control." := "dbHold_Sending".data."Time".Start_przetłaczanie_1.MINUTE)
      "Saving_Canged_Data_Word_USInt"("dbHold_download.sterowanie" := "dbHold_download".SendingTimes.Start_przetłaczanie_1.MINUTE, "DB10_instance_SCADA." := "DB10_instance_SCADA".actDTL_pumpingOn.MINUTE, memTrig_Client_Receiving_ := "memTrig_Client_Receiving_10")
   END_RUNG
   // the same network as SCL:
   "Detection_Changes_Data_Word_USInt"("tempdbHold_SendingTCP.sterowanie." := "tempdbHold_SendingTCP".Start_przetłaczanie_1.MINUTE,
                           "DB10_instance_SCADA." := "DB10_instance_SCADA".actDTL_pumpingOn.MINUTE,
                           memRisingTriger_Data_ := "memRisingTriger_Data_10",
                           "dbHold_Sending.data.stat.control." := "dbHold_Sending".data."Time".Start_przetłaczanie_1.MINUTE,
                           ENO => #_w1);
   IF #_w1 THEN
       "Saving_Canged_Data_Word_USInt"("dbHold_download.sterowanie" := "dbHold_download".SendingTimes.Start_przetłaczanie_1.MINUTE,
                               "DB10_instance_SCADA." := "DB10_instance_SCADA".actDTL_pumpingOn.MINUTE,
                               memTrig_Client_Receiving_ := "memTrig_Client_Receiving_10");
   END_IF;
END_REGION

REGION Network 12: Stop przetłaczanie (miasto) godziny
   RUNG wire#powerrail
      "Detection_Changes_Data_Word_USInt"("tempdbHold_SendingTCP.sterowanie." := "tempdbHold_SendingTCP".Stop_przetłaczanie_1.HOUR, "DB10_instance_SCADA." := "DB10_instance_SCADA".actDTL_pumpingOff.HOUR, memRisingTriger_Data_ := "memRisingTriger_Data_11", "dbHold_Sending.data.stat.control." := "dbHold_Sending".data."Time".Stop_przetłaczanie_1.HOUR)
      "Saving_Canged_Data_Word_USInt"("dbHold_download.sterowanie" := "dbHold_download".SendingTimes.Stop_przetłaczanie_1.HOUR, "DB10_instance_SCADA." := "DB10_instance_SCADA".actDTL_pumpingOff.HOUR, memTrig_Client_Receiving_ := "memTrig_Client_Receiving_11")
   END_RUNG
   // the same network as SCL:
   "Detection_Changes_Data_Word_USInt"("tempdbHold_SendingTCP.sterowanie." := "tempdbHold_SendingTCP".Stop_przetłaczanie_1.HOUR,
                           "DB10_instance_SCADA." := "DB10_instance_SCADA".actDTL_pumpingOff.HOUR,
                           memRisingTriger_Data_ := "memRisingTriger_Data_11",
                           "dbHold_Sending.data.stat.control." := "dbHold_Sending".data."Time".Stop_przetłaczanie_1.HOUR,
                           ENO => #_w1);
   IF #_w1 THEN
       "Saving_Canged_Data_Word_USInt"("dbHold_download.sterowanie" := "dbHold_download".SendingTimes.Stop_przetłaczanie_1.HOUR,
                               "DB10_instance_SCADA." := "DB10_instance_SCADA".actDTL_pumpingOff.HOUR,
                               memTrig_Client_Receiving_ := "memTrig_Client_Receiving_11");
   END_IF;
END_REGION

REGION Network 13: Stop przetłaczanie (miasto) minuty
   RUNG wire#powerrail
      "Detection_Changes_Data_Word_USInt"("tempdbHold_SendingTCP.sterowanie." := "tempdbHold_SendingTCP".Stop_przetłaczanie_1.MINUTE, "DB10_instance_SCADA." := "DB10_instance_SCADA".actDTL_pumpingOff.MINUTE, memRisingTriger_Data_ := "memRisingTriger_Data_12", "dbHold_Sending.data.stat.control." := "dbHold_Sending".data."Time".Stop_przetłaczanie_1.MINUTE)
      "Saving_Canged_Data_Word_USInt"("dbHold_download.sterowanie" := "dbHold_download".SendingTimes.Stop_przetłaczanie_1.MINUTE, "DB10_instance_SCADA." := "DB10_instance_SCADA".actDTL_pumpingOff.MINUTE, memTrig_Client_Receiving_ := "memTrig_Client_Receiving_12")
   END_RUNG
   // the same network as SCL:
   "Detection_Changes_Data_Word_USInt"("tempdbHold_SendingTCP.sterowanie." := "tempdbHold_SendingTCP".Stop_przetłaczanie_1.MINUTE,
                           "DB10_instance_SCADA." := "DB10_instance_SCADA".actDTL_pumpingOff.MINUTE,
                           memRisingTriger_Data_ := "memRisingTriger_Data_12",
                           "dbHold_Sending.data.stat.control." := "dbHold_Sending".data."Time".Stop_przetłaczanie_1.MINUTE,
                           ENO => #_w1);
   IF #_w1 THEN
       "Saving_Canged_Data_Word_USInt"("dbHold_download.sterowanie" := "dbHold_download".SendingTimes.Stop_przetłaczanie_1.MINUTE,
                               "DB10_instance_SCADA." := "DB10_instance_SCADA".actDTL_pumpingOff.MINUTE,
                               memTrig_Client_Receiving_ := "memTrig_Client_Receiving_12");
   END_IF;
END_REGION

REGION Network 14: Start dosilanie godziny
   RUNG wire#powerrail
      "Detection_Changes_Data_Word_USInt"("tempdbHold_SendingTCP.sterowanie." := "tempdbHold_SendingTCP".Start_dosilanie_1.HOUR, "DB10_instance_SCADA." := "DB10_instance_SCADA".actDTL_RechargingOn.HOUR, memRisingTriger_Data_ := "memRisingTriger_Data_13", "dbHold_Sending.data.stat.control." := "dbHold_Sending".data."Time".Start_dosilanie_1.HOUR)
      "Saving_Canged_Data_Word_USInt"("dbHold_download.sterowanie" := "dbHold_download".SendingTimes.Start_dosilanie_1.HOUR, "DB10_instance_SCADA." := "DB10_instance_SCADA".actDTL_RechargingOn.HOUR, memTrig_Client_Receiving_ := "memTrig_Client_Receiving_13")
   END_RUNG
   // the same network as SCL:
   "Detection_Changes_Data_Word_USInt"("tempdbHold_SendingTCP.sterowanie." := "tempdbHold_SendingTCP".Start_dosilanie_1.HOUR,
                           "DB10_instance_SCADA." := "DB10_instance_SCADA".actDTL_RechargingOn.HOUR,
                           memRisingTriger_Data_ := "memRisingTriger_Data_13",
                           "dbHold_Sending.data.stat.control." := "dbHold_Sending".data."Time".Start_dosilanie_1.HOUR,
                           ENO => #_w1);
   IF #_w1 THEN
       "Saving_Canged_Data_Word_USInt"("dbHold_download.sterowanie" := "dbHold_download".SendingTimes.Start_dosilanie_1.HOUR,
                               "DB10_instance_SCADA." := "DB10_instance_SCADA".actDTL_RechargingOn.HOUR,
                               memTrig_Client_Receiving_ := "memTrig_Client_Receiving_13");
   END_IF;
END_REGION

